C07322=1185.317,71.605,-48.992,-179.176,5.973,148.824
C07323=1185.312,71.854,-49.010,-179.174,5.974,148.823
C07324=1185.308,72.103,-49.027,-179.172,5.975,148.823
C07325=1185.303,72.353,-49.044,-179.168,5.976,148.822
C07326=1185.298,72.602,-49.061,-179.166,5.977,148.822
C07327=1185.293,72.852,-49.078,-179.163,5.978,148.821
C07328=1185.288,73.101,-49.095,-179.161,5.979,148.820
C07329=1185.283,73.350,-49.112,-179.158,5.980,148.820
C07330=1185.279,73.600,-49.129,-179.155,5.981,148.819
C07331=1185.273,73.849,-49.146,-179.153,5.982,148.819
C07332=1185.268,74.098,-49.163,-179.150,5.983,148.818
C07333=1185.263,74.347,-49.181,-179.148,5.984,148.818
C07334=1185.259,74.597,-49.197,-179.145,5.985,148.817
C07335=1185.254,74.847,-49.215,-179.143,5.986,148.817
C07336=1185.249,75.096,-49.231,-179.140,5.987,148.816
C07337=1185.244,75.345,-49.249,-179.137,5.988,148.815
C07338=1185.239,75.594,-49.266,-179.134,5.989,148.815
C07339=1185.234,75.844,-49.283,-179.132,5.990,148.814
C07340=1185.229,76.093,-49.301,-179.129,5.991,148.814
C07341=1185.225,76.343,-49.318,-179.127,5.992,148.813
C07342=1185.219,76.592,-49.335,-179.124,5.993,148.813
C07343=1185.215,76.842,-49.353,-179.122,5.994,148.812
C07344=1185.209,77.090,-49.369,-179.119,5.995,148.812
C07345=1185.205,77.340,-49.387,-179.116,5.996,148.811
C07346=1185.199,77.589,-49.404,-179.113,5.998,148.810
C07347=1185.195,77.839,-49.421,-179.111,5.998,148.810
C07348=1185.190,78.088,-49.439,-179.109,5.999,148.809
C07349=1185.185,78.337,-49.456,-179.105,6.000,148.809
C07350=1185.181,78.587,-49.474,-179.103,6.001,148.808
C07351=1185.175,78.836,-49.491,-179.101,6.002,148.808
C07352=1185.169,79.086,-49.508,-179.098,6.003,148.807
C07353=1185.165,79.334,-49.525,-179.095,6.004,148.807
C07354=1185.160,79.584,-49.542,-179.093,6.006,148.806
C07355=1185.155,79.833,-49.560,-179.090,6.006,148.805
C07356=1185.151,80.083,-49.577,-179.088,6.007,148.805
C07357=1185.146,80.351,-49.596,-179.085,6.009,148.804
C07358=1185.140,80.620,-49.615,-179.081,6.010,148.804
C07359=1185.134,80.888,-49.633,-179.079,6.011,148.803
C07360=1185.129,81.156,-49.653,-179.076,6.012,148.803
C07361=1185.125,81.406,-49.670,-179.073,6.013,148.802
C07362=1185.120,81.655,-49.688,-179.071,6.014,148.802
C07363=1185.115,81.905,-49.705,-179.068,6.015,148.801
C07364=1185.110,82.154,-49.723,-179.066,6.016,148.801
C07365=1185.105,82.403,-49.740,-179.063,6.017,148.800
C07366=1185.100,82.653,-49.757,-179.061,6.018,148.799
C07367=1185.095,82.902,-49.775,-179.057,6.019,148.799
C07368=1185.090,83.152,-49.793,-179.055,6.020,148.798
C07369=1185.086,83.401,-49.810,-179.053,6.021,148.798
C07370=1185.081,83.650,-49.828,-179.050,6.023,148.797
C07371=1185.076,83.900,-49.845,-179.047,6.023,148.797
C07372=1185.071,84.149,-49.863,-179.045,6.025,148.796
C07373=1185.066,84.398,-49.881,-179.042,6.025,148.796
C07374=1185.062,84.647,-49.898,-179.039,6.027,148.795
C07375=1185.057,84.897,-49.916,-179.037,6.028,148.795
C07376=1185.052,85.146,-49.934,-179.034,6.029,148.794
C07377=1185.046,85.396,-49.951,-179.032,6.030,148.794
C07378=1185.042,85.645,-49.969,-179.029,6.031,148.793
C07379=1185.037,85.894,-49.987,-179.026,6.033,148.793
C07380=1185.031,86.144,-50.004,-179.024,6.033,148.792
C07381=1185.027,86.393,-50.022,-179.021,6.035,148.792
C07382=1185.022,86.642,-50.040,-179.018,6.035,148.791
C07383=1185.017,86.891,-50.058,-179.016,6.036,148.790
C07384=1185.012,87.141,-50.075,-179.013,6.038,148.790
C07385=1185.007,87.390,-50.093,-179.011,6.039,148.789
C07386=1185.002,87.639,-50.111,-179.008,6.040,148.789
C07387=1184.997,87.888,-50.129,-179.006,6.041,148.788
C07388=1184.992,88.138,-50.146,-179.002,6.042,148.788
C07389=1184.987,88.387,-50.164,-179.000,6.043,148.787
C07390=1184.982,88.636,-50.182,-178.997,6.044,148.787
C07391=1184.978,88.885,-50.200,-178.995,6.045,148.786
C07392=1184.973,89.134,-50.218,-178.992,6.047,148.786
C07393=1184.968,89.384,-50.235,-178.990,6.048,148.785
C07394=1184.963,89.633,-50.253,-178.987,6.048,148.784
C07395=1184.958,89.883,-50.271,-178.984,6.050,148.784
C07396=1184.954,90.132,-50.289,-178.982,6.050,148.783
C07397=1184.949,90.382,-50.307,-178.979,6.052,148.783
C07398=1184.944,90.631,-50.325,-178.977,6.053,148.783
C07399=1184.939,90.880,-50.343,-178.974,6.054,148.782
C07400=1184.934,91.129,-50.361,-178.971,6.055,148.781
C07401=1184.929,91.378,-50.379,-178.968,6.057,148.781
C07402=1184.924,91.628,-50.396,-178.966,6.058,148.780
C07403=1184.919,91.877,-50.414,-178.963,6.059,148.780
C07404=1184.914,92.126,-50.432,-178.961,6.060,148.779
C07405=1184.910,92.376,-50.451,-178.958,6.061,148.779
C07406=1184.905,92.625,-50.469,-178.955,6.062,148.778
C07407=1184.900,92.875,-50.487,-178.953,6.063,148.778
C07408=1184.895,93.124,-50.505,-178.950,6.065,148.777
C07409=1184.890,93.373,-50.522,-178.948,6.065,148.777
C07410=1184.886,93.622,-50.540,-178.945,6.067,148.776
C07411=1184.880,93.872,-50.559,-178.943,6.068,148.776
C07412=1184.876,94.122,-50.577,-178.939,6.069,148.775
C07413=1184.871,94.371,-50.595,-178.937,6.070,148.775
C07414=1184.866,94.620,-50.613,-178.934,6.071,148.774
C07415=1184.861,94.869,-50.631,-178.932,6.072,148.774
C07416=1184.856,95.118,-50.649,-178.929,6.074,148.773
C07417=1184.851,95.367,-50.667,-178.927,6.075,148.773
C07418=1184.847,95.617,-50.686,-178.924,6.076,148.772
C07419=1184.842,95.866,-50.704,-178.921,6.077,148.771
C07420=1184.836,96.115,-50.723,-178.919,6.079,148.771
C07421=1184.832,96.365,-50.741,-178.916,6.079,148.770
C07422=1184.827,96.614,-50.759,-178.913,6.081,148.770
C07423=1184.822,96.864,-50.777,-178.911,6.081,148.769
C07424=1184.817,97.113,-50.795,-178.908,6.083,148.769
C07425=1184.812,97.362,-50.813,-178.905,6.084,148.768
C07426=1184.808,97.610,-50.832,-178.903,6.085,148.768
C07427=1184.802,97.860,-50.850,-178.900,6.086,148.767
C07428=1184.798,98.110,-50.869,-178.897,6.088,148.767
C07429=1184.793,98.359,-50.887,-178.895,6.089,148.766
C07430=1184.788,98.608,-50.905,-178.892,6.090,148.766
C07431=1184.783,98.857,-50.923,-178.890,6.091,148.765
C07432=1184.778,99.107,-50.942,-178.887,6.092,148.765
C07433=1184.774,99.356,-50.960,-178.884,6.093,148.764
C07434=1184.769,99.605,-50.978,-178.882,6.095,148.764
C07435=1184.764,99.854,-50.996,-178.879,6.095,148.763
C07436=1184.759,100.104,-51.016,-178.876,6.097,148.763
C07437=1184.754,100.353,-51.034,-178.873,6.099,148.762
C07438=1184.749,100.602,-51.052,-178.871,6.099,148.762
C07439=1184.744,100.852,-51.070,-178.868,6.101,148.761
C07440=1184.739,101.101,-51.090,-178.866,6.102,148.761
C07441=1184.735,101.350,-51.108,-178.863,6.104,148.760
C07442=1184.730,101.599,-51.126,-178.860,6.104,148.760
C07443=1184.726,101.849,-51.145,-178.858,6.106,148.759
C07444=1184.720,102.098,-51.163,-178.856,6.107,148.759
C07445=1184.715,102.347,-51.181,-178.852,6.108,148.758
C07446=1184.711,102.597,-51.200,-178.850,6.109,148.758
C07447=1184.705,102.846,-51.219,-178.847,6.110,148.757
C07448=1184.701,103.095,-51.237,-178.845,6.111,148.757
C07449=1184.696,103.344,-51.255,-178.842,6.113,148.756
C07450=1184.691,103.594,-51.274,-178.839,6.114,148.756
C07451=1184.686,103.843,-51.293,-178.837,6.115,148.755
C07452=1184.681,104.092,-51.311,-178.834,6.117,148.755
C07453=1184.676,104.342,-51.330,-178.832,6.118,148.754
C07454=1184.672,104.591,-51.349,-178.829,6.119,148.754
C07455=1184.667,104.840,-51.367,-178.826,6.120,148.753
C07456=1184.662,105.089,-51.386,-178.824,6.122,148.753
C07457=1184.657,105.338,-51.404,-178.821,6.122,148.752
C07458=1184.653,105.588,-51.423,-178.818,6.124,148.752
C07459=1184.647,105.837,-51.442,-178.816,6.125,148.751
C07460=1184.643,106.086,-51.461,-178.813,6.126,148.751
C07461=1184.638,106.355,-51.481,-178.810,6.128,148.750
C07462=1184.633,106.623,-51.501,-178.807,6.129,148.750
C07463=1184.627,106.891,-51.521,-178.804,6.130,148.749
C07464=1184.622,107.160,-51.542,-178.802,6.132,148.749
C07465=1184.617,107.409,-51.560,-178.799,6.133,148.748
C07466=1184.612,107.659,-51.579,-178.796,6.134,148.748
C07467=1184.608,107.908,-51.598,-178.794,6.136,148.747
C07468=1184.603,108.156,-51.617,-178.791,6.136,148.746
C07469=1184.598,108.407,-51.636,-178.788,6.138,148.746
C07470=1184.593,108.655,-51.654,-178.786,6.140,148.746
C07471=1184.588,108.905,-51.673,-178.783,6.140,148.745
C07472=1184.584,109.154,-51.692,-178.780,6.142,148.745
C07473=1184.578,109.403,-51.711,-178.778,6.143,148.744
C07474=1184.574,109.653,-51.729,-178.775,6.144,148.744
C07475=1184.569,109.901,-51.749,-178.773,6.145,148.743
C07476=1184.565,110.151,-51.768,-178.770,6.147,148.743
C07477=1184.559,110.400,-51.786,-178.767,6.148,148.742
C07478=1184.554,110.649,-51.805,-178.765,6.149,148.742
C07479=1184.550,110.898,-51.825,-178.762,6.151,148.741
C07480=1184.545,111.147,-51.843,-178.759,6.152,148.741
C07481=1184.540,111.397,-51.862,-178.757,6.153,148.740
C07482=1184.535,111.646,-51.882,-178.754,6.155,148.740
C07483=1184.530,111.896,-51.900,-178.751,6.156,148.739
C07484=1184.525,112.145,-51.919,-178.749,6.157,148.739
C07485=1184.521,112.394,-51.938,-178.746,6.158,148.738
C07486=1184.516,112.643,-51.958,-178.743,6.160,148.738
C07487=1184.511,112.893,-51.976,-178.741,6.161,148.737
C07488=1184.506,113.142,-51.995,-178.738,6.162,148.737
C07489=1184.501,113.391,-52.015,-178.735,6.164,148.736
C07490=1184.497,113.640,-52.034,-178.733,6.164,148.736
C07491=1184.492,113.889,-52.053,-178.730,6.166,148.735
C07492=1184.487,114.138,-52.071,-178.727,6.168,148.735
C07493=1184.482,114.388,-52.091,-178.725,6.168,148.734
C07494=1184.477,114.637,-52.110,-178.722,6.170,148.734
C07495=1184.473,114.886,-52.129,-178.719,6.172,148.733
C07496=1184.468,115.135,-52.149,-178.717,6.172,148.733
C07497=1184.463,115.385,-52.168,-178.714,6.174,148.732
C07498=1184.458,115.634,-52.186,-178.712,6.175,148.732
C07499=1184.453,115.883,-52.206,-178.709,6.176,148.731
C07500=1184.448,116.132,-52.225,-178.706,6.178,148.731
C07501=1184.444,116.381,-52.244,-178.704,6.179,148.731
C07502=1184.438,116.630,-52.264,-178.701,6.181,148.730
C07503=1184.434,116.880,-52.283,-178.698,6.182,148.730
C07504=1184.428,117.129,-52.302,-178.696,6.183,148.729
C07505=1184.424,117.378,-52.322,-178.693,6.185,148.729
C07506=1184.420,117.628,-52.341,-178.691,6.185,148.728
C07507=1184.414,117.876,-52.360,-178.688,6.187,148.728
C07508=1184.410,118.126,-52.380,-178.685,6.189,148.727
C07509=1184.405,118.375,-52.399,-178.683,6.190,148.727
C07510=1184.400,118.624,-52.418,-178.680,6.191,148.726
C07511=1184.395,118.874,-52.438,-178.677,6.193,148.726
C07512=1184.391,119.122,-52.457,-178.675,6.194,148.725
C07513=1184.386,119.372,-52.476,-178.672,6.195,148.725
C07514=1184.381,119.621,-52.496,-178.669,6.197,148.724
C07515=1184.376,119.870,-52.515,-178.667,6.198,148.724
C07516=1184.371,120.120,-52.535,-178.664,6.199,148.723
C07517=1184.367,120.368,-52.554,-178.661,6.201,148.723
C07518=1184.362,120.618,-52.573,-178.658,6.202,148.722
C07519=1184.357,120.867,-52.593,-178.656,6.203,148.722
C07520=1184.352,121.116,-52.612,-178.653,6.205,148.722
C07521=1184.347,121.366,-52.632,-178.650,6.206,148.721
C07522=1184.343,121.614,-52.651,-178.648,6.208,148.721
C07523=1184.338,121.863,-52.671,-178.645,6.209,148.720
C07524=1184.333,122.113,-52.691,-178.643,6.210,148.720
C07525=1184.328,122.362,-52.710,-178.640,6.212,148.719
C07526=1184.323,122.611,-52.730,-178.637,6.213,148.719
C07527=1184.318,122.861,-52.749,-178.635,6.214,148.718
C07528=1184.313,123.110,-52.769,-178.632,6.216,148.718
C07529=1184.309,123.358,-52.788,-178.629,6.217,148.717
C07530=1184.305,123.608,-52.808,-178.627,6.218,148.717
C07531=1184.299,123.857,-52.827,-178.624,6.220,148.716
C07532=1184.295,124.106,-52.847,-178.621,6.221,148.716
C07533=1184.290,124.355,-52.867,-178.619,6.222,148.715
C07534=1184.285,124.604,-52.887,-178.616,6.224,148.715
C07535=1184.280,124.854,-52.906,-178.613,6.226,148.714
C07536=1184.275,125.103,-52.926,-178.611,6.226,148.714
C07537=1184.271,125.352,-52.946,-178.608,6.228,148.714
C07538=1184.266,125.601,-52.966,-178.606,6.230,148.713
C07539=1184.261,125.851,-52.985,-178.603,6.231,148.713
C07540=1184.256,126.100,-53.005,-178.600,6.232,148.712
C07541=1184.252,126.348,-53.024,-178.598,6.234,148.712
C07542=1184.247,126.598,-53.044,-178.595,6.235,148.711
C07543=1184.242,126.847,-53.064,-178.592,6.236,148.711
C07544=1184.238,127.096,-53.084,-178.590,6.238,148.710
C07545=1184.232,127.345,-53.103,-178.587,6.240,148.710
C07546=1184.228,127.595,-53.123,-178.584,6.240,148.709
C07547=1184.223,127.844,-53.143,-178.582,6.242,148.709
C07548=1184.219,128.093,-53.163,-178.579,6.244,148.709
C07549=1184.214,128.342,-53.183,-178.577,6.245,148.708
C07550=1184.209,128.591,-53.203,-178.574,6.246,148.708
C07551=1184.204,128.841,-53.222,-178.571,6.248,148.707
C07552=1184.200,129.090,-53.243,-178.568,6.250,148.707
C07553=1184.194,129.340,-53.263,-178.566,6.251,148.706
C07554=1184.189,129.588,-53.283,-178.563,6.252,148.706
C07555=1184.184,129.837,-53.303,-178.560,6.254,148.705
C07556=1184.180,130.086,-53.323,-178.558,6.255,148.705
C07557=1184.175,130.336,-53.343,-178.555,6.257,148.705
C07558=1184.171,130.585,-53.363,-178.552,6.258,148.704
C07559=1184.165,130.834,-53.382,-178.549,6.260,148.704
C07560=1184.161,131.083,-53.403,-178.547,6.261,148.703
C07561=1184.156,131.332,-53.422,-178.545,6.262,148.703
C07562=1184.152,131.581,-53.443,-178.541,6.264,148.702
C07563=1184.147,131.831,-53.462,-178.539,6.265,148.702
C07564=1184.141,132.079,-53.483,-178.537,6.266,148.701
C07565=1184.136,132.348,-53.504,-178.533,6.268,148.701
C07566=1184.131,132.618,-53.526,-178.531,6.270,148.700
C07567=1184.127,132.886,-53.548,-178.528,6.271,148.700
C07568=1184.121,133.155,-53.570,-178.525,6.273,148.699
C07569=1184.116,133.403,-53.590,-178.522,6.275,148.699
C07570=1184.111,133.652,-53.609,-178.519,6.276,148.699
C07571=1184.107,133.901,-53.630,-178.517,6.277,148.698
C07572=1184.102,134.150,-53.650,-178.514,6.279,148.698
C07573=1184.098,134.400,-53.670,-178.511,6.280,148.697
C07574=1184.092,134.649,-53.691,-178.509,6.281,148.697
C07575=1184.088,134.898,-53.711,-178.507,6.283,148.696
C07576=1184.083,135.148,-53.731,-178.503,6.284,148.696
C07577=1184.078,135.396,-53.751,-178.501,6.286,148.695
C07578=1184.073,135.645,-53.772,-178.498,6.288,148.695
C07579=1184.068,135.895,-53.791,-178.496,6.289,148.695
C07580=1184.064,136.144,-53.812,-178.493,6.291,148.694
C07581=1184.059,136.393,-53.832,-178.490,6.292,148.694
C07582=1184.054,136.642,-53.853,-178.487,6.294,148.693
C07583=1184.050,136.891,-53.873,-178.485,6.295,148.693
C07584=1184.045,137.140,-53.893,-178.483,6.297,148.692
C07585=1184.041,137.389,-53.913,-178.479,6.298,148.692
C07586=1184.035,137.639,-53.934,-178.477,6.300,148.691
C07587=1184.031,137.888,-53.955,-178.475,6.301,148.691
C07588=1184.026,138.137,-53.974,-178.472,6.302,148.691
C07589=1184.022,138.386,-53.995,-178.469,6.304,148.690
C07590=1184.016,138.635,-54.015,-178.466,6.306,148.690
C07591=1184.012,138.884,-54.036,-178.464,6.306,148.689
C07592=1184.007,139.133,-54.056,-178.461,6.308,148.689
C07593=1184.002,139.382,-54.077,-178.459,6.310,148.688
C07594=1183.997,139.631,-54.097,-178.456,6.312,148.688
C07595=1183.993,139.880,-54.117,-178.453,6.313,148.687
C07596=1183.988,140.130,-54.138,-178.451,6.314,148.687
C07597=1183.983,140.379,-54.158,-178.448,6.316,148.687
C07598=1183.978,140.628,-54.179,-178.445,6.318,148.686
C07599=1183.974,140.877,-54.200,-178.442,6.319,148.686
C07600=1183.969,141.126,-54.220,-178.440,6.321,148.686
C07601=1183.964,141.375,-54.241,-178.437,6.322,148.685
C07602=1183.960,141.624,-54.262,-178.434,6.323,148.684
C07603=1183.955,141.873,-54.282,-178.432,6.325,148.684
C07604=1183.950,142.122,-54.303,-178.429,6.327,148.684
C07605=1183.946,142.371,-54.323,-178.426,6.329,148.683
C07606=1183.940,142.620,-54.344,-178.424,6.329,148.683
C07607=1183.936,142.869,-54.365,-178.421,6.331,148.682
C07608=1183.931,143.119,-54.386,-178.418,6.333,148.682
C07609=1183.926,143.367,-54.406,-178.416,6.335,148.682
C07610=1183.922,143.616,-54.426,-178.413,6.336,148.681
C07611=1183.917,143.866,-54.448,-178.411,6.337,148.681
C07612=1183.913,144.115,-54.468,-178.408,6.339,148.680
C07613=1183.908,144.365,-54.489,-178.405,6.341,148.680
C07614=1183.903,144.614,-54.509,-178.402,6.342,148.679
C07615=1183.898,144.863,-54.530,-178.400,6.344,148.679
C07616=1183.894,145.112,-54.551,-178.397,6.346,148.679
C07617=1183.888,145.361,-54.572,-178.395,6.347,148.678
C07618=1183.884,145.610,-54.592,-178.392,6.348,148.678
C07619=1183.879,145.859,-54.613,-178.389,6.350,148.677
C07620=1183.875,146.108,-54.634,-178.386,6.352,148.677
C07621=1183.870,146.357,-54.655,-178.384,6.353,148.676
C07622=1183.865,146.606,-54.675,-178.382,6.354,148.676
C07623=1183.860,146.855,-54.696,-178.379,6.356,148.676
C07624=1183.855,147.105,-54.718,-178.376,6.358,148.675
C07625=1183.851,147.354,-54.738,-178.373,6.359,148.675
C07626=1183.846,147.603,-54.760,-178.370,6.361,148.674
C07627=1183.842,147.852,-54.780,-178.368,6.363,148.674
C07628=1183.836,148.101,-54.801,-178.365,6.364,148.674
C07629=1183.832,148.350,-54.821,-178.363,6.366,148.673
C07630=1183.827,148.598,-54.843,-178.360,6.367,148.673
C07631=1183.822,148.848,-54.864,-178.357,6.369,148.672
C07632=1183.818,149.097,-54.885,-178.355,6.371,148.672
C07633=1183.813,149.347,-54.906,-178.352,6.372,148.671
C07634=1183.809,149.595,-54.927,-178.349,6.374,148.671
C07635=1183.804,149.844,-54.948,-178.347,6.375,148.671
C07636=1183.798,150.093,-54.969,-178.344,6.377,148.670
C07637=1183.794,150.342,-54.990,-178.341,6.378,148.670
C07638=1183.790,150.592,-55.011,-178.339,6.380,148.670
C07639=1183.785,150.841,-55.032,-178.336,6.382,148.669
C07640=1183.780,151.089,-55.053,-178.333,6.384,148.669
C07641=1183.775,151.339,-55.074,-178.330,6.385,148.668
C07642=1183.770,151.588,-55.095,-178.328,6.386,148.668
C07643=1183.765,151.836,-55.117,-178.325,6.388,148.667
C07644=1183.761,152.086,-55.138,-178.323,6.390,148.667
C07645=1183.757,152.335,-55.159,-178.320,6.391,148.667
C07646=1183.751,152.584,-55.180,-178.317,6.393,148.666
C07647=1183.747,152.833,-55.201,-178.315,6.395,148.666
C07648=1183.742,153.082,-55.222,-178.312,6.397,148.666
C07649=1183.737,153.332,-55.244,-178.309,6.399,148.665
C07650=1183.733,153.580,-55.265,-178.307,6.399,148.665
C07651=1183.728,153.829,-55.286,-178.304,6.401,148.664
C07652=1183.723,154.078,-55.307,-178.301,6.403,148.664
C07653=1183.719,154.328,-55.329,-178.299,6.404,148.663
C07654=1183.714,154.576,-55.350,-178.296,6.406,148.663
C07655=1183.709,154.825,-55.371,-178.293,6.408,148.663
C07656=1183.705,155.074,-55.393,-178.291,6.410,148.662
C07657=1183.700,155.324,-55.414,-178.288,6.411,148.662
C07658=1183.695,155.573,-55.436,-178.285,6.413,148.662
C07659=1183.690,155.822,-55.456,-178.283,6.414,148.661
C07660=1183.686,156.070,-55.478,-178.280,6.416,148.661
C07661=1183.682,156.319,-55.500,-178.277,6.417,148.660
C07662=1183.676,156.569,-55.521,-178.275,6.419,148.660
C07663=1183.671,156.817,-55.542,-178.272,6.421,148.659
C07664=1183.667,157.067,-55.564,-178.269,6.423,148.659
C07665=1183.662,157.316,-55.585,-178.266,6.424,148.659
C07666=1183.657,157.565,-55.607,-178.264,6.426,148.658
C07667=1183.653,157.814,-55.627,-178.261,6.428,148.658
C07668=1183.648,158.063,-55.649,-178.258,6.430,148.658
C07669=1183.643,158.332,-55.673,-178.256,6.432,148.657
C07670=1183.638,158.601,-55.696,-178.253,6.433,148.657
C07671=1183.633,158.870,-55.720,-178.250,6.435,148.656
C07672=1183.628,159.138,-55.742,-178.247,6.436,148.656
C07673=1183.623,159.388,-55.764,-178.245,6.438,148.655
C07674=1183.618,159.637,-55.785,-178.242,6.440,148.655
C07675=1183.613,159.886,-55.807,-178.239,6.442,148.655
C07676=1183.609,160.135,-55.829,-178.236,6.444,148.654
C07677=1183.604,160.384,-55.850,-178.234,6.445,148.654
C07678=1183.600,160.634,-55.872,-178.231,6.447,148.654
C07679=1183.595,160.882,-55.893,-178.228,6.449,148.653
C07680=1183.590,161.131,-55.915,-178.225,6.450,148.653
C07681=1183.586,161.380,-55.937,-178.223,6.451,148.652
C07682=1183.581,161.629,-55.959,-178.220,6.453,148.652
C07683=1183.576,161.878,-55.980,-178.218,6.455,148.651
C07684=1183.571,162.127,-56.002,-178.215,6.457,148.651
C07685=1183.566,162.376,-56.024,-178.212,6.458,148.651
C07686=1183.562,162.625,-56.046,-178.210,6.460,148.650
C07687=1183.557,162.874,-56.067,-178.207,6.462,148.650
C07688=1183.552,163.123,-56.089,-178.204,6.464,148.650
C07689=1183.548,163.372,-56.111,-178.202,6.465,148.649
C07690=1183.543,163.621,-56.132,-178.199,6.467,148.649
C07691=1183.539,163.871,-56.154,-178.196,6.469,148.649
C07692=1183.534,164.119,-56.176,-178.194,6.471,148.648
C07693=1183.529,164.368,-56.197,-178.191,6.473,148.648
C07694=1183.525,164.617,-56.219,-178.188,6.474,148.647
C07695=1183.520,164.866,-56.241,-178.186,6.476,148.647
C07696=1183.516,165.115,-56.263,-178.183,6.478,148.647
C07697=1183.511,165.364,-56.285,-178.180,6.480,148.646
C07698=1183.506,165.613,-56.307,-178.178,6.481,148.646
C07699=1183.502,165.862,-56.329,-178.175,6.483,148.646
C07700=1183.497,166.112,-56.351,-178.173,6.484,148.645
C07701=1183.492,166.360,-56.373,-178.170,6.486,148.645
C07702=1183.487,166.610,-56.395,-178.167,6.488,148.644
C07703=1183.483,166.858,-56.417,-178.165,6.489,148.644
C07704=1183.478,167.108,-56.439,-178.162,6.491,148.644
C07705=1183.473,167.356,-56.460,-178.159,6.493,148.643
C07706=1183.469,167.605,-56.482,-178.157,6.495,148.643
C07707=1183.464,167.854,-56.505,-178.154,6.497,148.643
C07708=1183.459,168.102,-56.527,-178.151,6.498,148.642
C07709=1183.455,168.352,-56.549,-178.149,6.500,148.642
C07710=1183.450,168.600,-56.571,-178.146,6.502,148.641
C07711=1183.446,168.850,-56.593,-178.143,6.504,148.641
C07712=1183.441,169.099,-56.616,-178.141,6.505,148.641
C07713=1183.436,169.348,-56.637,-178.138,6.507,148.640
C07714=1183.431,169.597,-56.659,-178.135,6.509,148.640
C07715=1183.427,169.846,-56.681,-178.133,6.511,148.640
C07716=1183.423,170.095,-56.704,-178.130,6.513,148.639
C07717=1183.417,170.344,-56.726,-178.127,6.514,148.639
C07718=1183.413,170.593,-56.748,-178.125,6.516,148.639
C07719=1183.408,170.842,-56.770,-178.122,6.518,148.638
C07720=1183.404,171.091,-56.792,-178.119,6.520,148.638
C07721=1183.398,171.339,-56.815,-178.117,6.521,148.637
C07722=1183.394,171.589,-56.837,-178.114,6.523,148.637
C07723=1183.389,171.837,-56.858,-178.111,6.525,148.637
C07724=1183.385,172.086,-56.882,-178.108,6.527,148.636
C07725=1183.380,172.336,-56.904,-178.106,6.529,148.636
C07726=1183.375,172.584,-56.926,-178.103,6.530,148.636
C07727=1183.370,172.834,-56.948,-178.100,6.532,148.635
C07728=1183.366,173.082,-56.971,-178.098,6.534,148.635
C07729=1183.362,173.331,-56.993,-178.095,6.536,148.635
C07730=1183.357,173.581,-57.015,-178.092,6.537,148.634
C07731=1183.352,173.829,-57.038,-178.090,6.539,148.634
C07732=1183.348,174.078,-57.060,-178.087,6.541,148.633
C07733=1183.342,174.327,-57.082,-178.084,6.543,148.633
C07734=1183.338,174.576,-57.105,-178.082,6.545,148.633
C07735=1183.334,174.825,-57.127,-178.079,6.546,148.632
C07736=1183.329,175.074,-57.150,-178.076,6.548,148.632
C07737=1183.324,175.323,-57.172,-178.074,6.550,148.632
C07738=1183.319,175.573,-57.195,-178.071,6.552,148.631
C07739=1183.315,175.821,-57.217,-178.068,6.553,148.631
C07740=1183.310,176.070,-57.239,-178.066,6.555,148.631
C07741=1183.305,176.318,-57.262,-178.063,6.557,148.630
C07742=1183.301,176.568,-57.284,-178.060,6.560,148.630
C07743=1183.296,176.817,-57.307,-178.058,6.562,148.630
C07744=1183.291,177.065,-57.329,-178.055,6.564,148.629
C07745=1183.287,177.314,-57.352,-178.052,6.565,148.629
C07746=1183.282,177.564,-57.374,-178.050,6.567,148.629
C07747=1183.278,177.812,-57.397,-178.047,6.569,148.628
C07748=1183.273,178.061,-57.419,-178.044,6.571,148.628
C07749=1183.269,178.310,-57.442,-178.042,6.572,148.628
C07750=1183.264,178.560,-57.465,-178.039,6.574,148.627
C07751=1183.259,178.808,-57.487,-178.036,6.576,148.627
C07752=1183.255,179.057,-57.511,-178.033,6.578,148.626
C07753=1183.250,179.306,-57.533,-178.031,6.580,148.626
C07754=1183.245,179.555,-57.556,-178.028,6.581,148.626
C07755=1183.241,179.804,-57.578,-178.025,6.583,148.625
C07756=1183.236,180.053,-57.601,-178.023,6.585,148.625
C07757=1183.232,180.302,-57.624,-178.021,6.587,148.625
C07758=1183.226,180.551,-57.646,-178.018,6.589,148.625
C07759=1183.222,180.800,-57.669,-178.015,6.591,148.624
C07760=1183.218,181.048,-57.692,-178.013,6.592,148.624
C07761=1183.213,181.298,-57.715,-178.009,6.595,148.623
C07762=1183.208,181.546,-57.737,-178.007,6.597,148.623
C07763=1183.204,181.795,-57.761,-178.004,6.599,148.623
C07764=1183.199,182.044,-57.783,-178.001,6.600,148.622
C07765=1183.195,182.293,-57.806,-177.999,6.602,148.622
C07766=1183.189,182.542,-57.829,-177.996,6.604,148.622
C07767=1183.185,182.791,-57.852,-177.994,6.606,148.622
C07768=1183.180,183.040,-57.874,-177.991,6.608,148.621
C07769=1183.176,183.289,-57.897,-177.988,6.610,148.621
C07770=1183.172,183.538,-57.921,-177.986,6.611,148.620
C07771=1183.166,183.786,-57.944,-177.983,6.613,148.620
C07772=1183.162,184.035,-57.966,-177.980,6.615,148.620
C07773=1183.157,184.305,-57.991,-177.977,6.618,148.619
C07774=1183.152,184.575,-58.016,-177.975,6.619,148.619
C07775=1183.147,184.844,-58.041,-177.972,6.621,148.619
C07776=1183.142,185.114,-58.066,-177.969,6.624,148.618
C07777=1183.137,185.363,-58.089,-177.966,6.626,148.618
C07778=1183.133,185.611,-58.112,-177.963,6.627,148.618
C07779=1183.128,185.861,-58.135,-177.961,6.629,148.617
C07780=1183.123,186.109,-58.158,-177.958,6.631,148.617
C07781=1183.119,186.358,-58.180,-177.956,6.633,148.617
C07782=1183.114,186.607,-58.204,-177.953,6.635,148.616
C07783=1183.109,186.856,-58.227,-177.950,6.637,148.616
C07784=1183.105,187.105,-58.250,-177.947,6.639,148.616
C07785=1183.101,187.354,-58.273,-177.944,6.641,148.615
C07786=1183.096,187.603,-58.297,-177.942,6.643,148.615
C07787=1183.091,187.852,-58.320,-177.939,6.645,148.615
C07788=1183.086,188.100,-58.343,-177.936,6.646,148.614
C07789=1183.082,188.349,-58.366,-177.934,6.648,148.614
C07790=1183.077,188.598,-58.389,-177.932,6.650,148.614
C07791=1183.073,188.847,-58.412,-177.929,6.652,148.614
C07792=1183.068,189.096,-58.436,-177.926,6.655,148.613
C07793=1183.063,189.345,-58.459,-177.923,6.656,148.613
C07794=1183.059,189.594,-58.482,-177.920,6.658,148.613
C07795=1183.055,189.843,-58.505,-177.918,6.660,148.612
C07796=1183.050,190.091,-58.529,-177.915,6.662,148.612
C07797=1183.045,190.340,-58.552,-177.913,6.664,148.612
C07798=1183.040,190.589,-58.576,-177.910,6.666,148.611
C07799=1183.036,190.838,-58.599,-177.907,6.668,148.611
C07800=1183.031,191.087,-58.622,-177.904,6.670,148.611
C07801=1183.027,191.336,-58.645,-177.902,6.672,148.610
C07802=1183.022,191.585,-58.669,-177.899,6.674,148.610
C07803=1183.018,191.834,-58.692,-177.897,6.676,148.610
C07804=1183.013,192.082,-58.716,-177.894,6.678,148.609
C07805=1183.008,192.331,-58.739,-177.891,6.679,148.609
C07806=1183.004,192.580,-58.763,-177.888,6.682,148.609
C07807=1182.999,192.829,-58.786,-177.885,6.684,148.608
C07808=1182.994,193.078,-58.809,-177.883,6.686,148.608
C07809=1182.990,193.327,-58.833,-177.881,6.688,148.608
C07810=1182.985,193.576,-58.857,-177.878,6.690,148.608
C07811=1182.981,193.825,-58.880,-177.875,6.691,148.607
C07812=1182.976,194.074,-58.904,-177.873,6.693,148.607
C07813=1182.971,194.322,-58.928,-177.870,6.696,148.607
C07814=1182.967,194.571,-58.951,-177.867,6.698,148.606
C07815=1182.962,194.820,-58.974,-177.865,6.700,148.606
C07816=1182.958,195.069,-58.998,-177.862,6.701,148.606
C07817=1182.953,195.318,-59.022,-177.859,6.703,148.605
C07818=1182.948,195.567,-59.045,-177.857,6.705,148.605
C07819=1182.944,195.815,-59.069,-177.854,6.708,148.605
C07820=1182.939,196.064,-59.093,-177.851,6.710,148.605
C07821=1182.934,196.313,-59.116,-177.848,6.712,148.604
C07822=1182.930,196.562,-59.140,-177.846,6.713,148.604
C07823=1182.925,196.811,-59.163,-177.843,6.715,148.604
C07824=1182.921,197.060,-59.187,-177.841,6.717,148.603
C07825=1182.916,197.308,-59.211,-177.838,6.720,148.603
C07826=1182.912,197.557,-59.234,-177.835,6.722,148.603
C07827=1182.907,197.805,-59.258,-177.832,6.723,148.602
C07828=1182.902,198.054,-59.282,-177.830,6.725,148.602
C07829=1182.898,198.303,-59.306,-177.828,6.727,148.602
C07830=1182.893,198.552,-59.329,-177.824,6.730,148.602
C07831=1182.890,198.801,-59.353,-177.822,6.732,148.601
C07832=1182.885,199.050,-59.377,-177.819,6.734,148.601
C07833=1182.880,199.299,-59.402,-177.817,6.736,148.601
C07834=1182.875,199.548,-59.425,-177.814,6.738,148.600
C07835=1182.871,199.796,-59.449,-177.811,6.740,148.600
C07836=1182.866,200.045,-59.472,-177.808,6.742,148.600
C07837=1182.862,200.294,-59.496,-177.806,6.744,148.599
C07838=1182.857,200.543,-59.520,-177.803,6.746,148.599
C07839=1182.852,200.791,-59.544,-177.801,6.748,148.599
C07840=1182.848,201.041,-59.568,-177.797,6.750,148.599
C07841=1182.843,201.290,-59.592,-177.795,6.752,148.598
C07842=1182.839,201.538,-59.616,-177.793,6.754,148.598
C07843=1182.834,201.787,-59.640,-177.790,6.756,148.598
C07844=1182.830,202.035,-59.664,-177.787,6.758,148.597
C07845=1182.825,202.284,-59.688,-177.784,6.760,148.597
C07846=1182.820,202.533,-59.712,-177.782,6.763,148.597
C07847=1182.816,202.782,-59.736,-177.779,6.764,148.597
C07848=1182.812,203.031,-59.760,-177.777,6.766,148.596
C07849=1182.806,203.280,-59.784,-177.773,6.769,148.596
C07850=1182.802,203.528,-59.808,-177.771,6.771,148.596
C07851=1182.798,203.777,-59.832,-177.768,6.773,148.596
C07852=1182.793,204.026,-59.856,-177.766,6.775,148.595
C07853=1182.788,204.275,-59.881,-177.763,6.776,148.595
C07854=1182.784,204.524,-59.905,-177.760,6.779,148.595
C07855=1182.780,204.772,-59.929,-177.758,6.781,148.594
C07856=1182.775,205.021,-59.953,-177.755,6.783,148.594
C07857=1182.770,205.270,-59.977,-177.752,6.785,148.594
C07858=1182.766,205.519,-60.001,-177.750,6.788,148.594
C07859=1182.761,205.767,-60.025,-177.747,6.789,148.593
C07860=1182.756,206.016,-60.050,-177.744,6.791,148.593
C07861=1182.752,206.265,-60.074,-177.742,6.793,148.593
C07862=1182.748,206.514,-60.098,-177.739,6.796,148.593
C07863=1182.743,206.763,-60.123,-177.736,6.798,148.592
C07864=1182.738,207.011,-60.147,-177.734,6.800,148.592
C07865=1182.734,207.260,-60.171,-177.731,6.802,148.592
C07866=1182.729,207.509,-60.196,-177.728,6.804,148.591
C07867=1182.725,207.758,-60.220,-177.725,6.806,148.591
C07868=1182.720,208.006,-60.245,-177.723,6.808,148.591
C07869=1182.716,208.255,-60.269,-177.721,6.810,148.591
C07870=1182.712,208.504,-60.293,-177.717,6.813,148.590
C07871=1182.706,208.753,-60.317,-177.715,6.814,148.590
C07872=1182.702,209.002,-60.341,-177.713,6.817,148.590
C07873=1182.697,209.250,-60.366,-177.710,6.818,148.589
C07874=1182.693,209.500,-60.390,-177.707,6.821,148.589
C07875=1182.688,209.748,-60.415,-177.705,6.823,148.589
C07876=1182.683,209.997,-60.439,-177.702,6.825,148.589
C07877=1182.679,210.268,-60.466,-177.699,6.828,148.588
C07878=1182.674,210.538,-60.493,-177.696,6.829,148.588
C07879=1182.669,210.808,-60.519,-177.693,6.832,148.588
C07880=1182.663,211.078,-60.546,-177.690,6.834,148.587
C07881=1182.660,211.327,-60.571,-177.687,6.837,148.587
C07882=1182.654,211.576,-60.595,-177.685,6.839,148.587
C07883=1182.650,211.824,-60.619,-177.682,6.840,148.587
C07884=1182.646,212.074,-60.644,-177.679,6.843,148.587
C07885=1182.641,212.322,-60.668,-177.677,6.845,148.586
C07886=1182.636,212.571,-60.693,-177.674,6.847,148.586
C07887=1182.632,212.820,-60.718,-177.672,6.849,148.586
C07888=1182.627,213.068,-60.743,-177.669,6.852,148.585
C07889=1182.624,213.317,-60.767,-177.666,6.854,148.585
C07890=1182.618,213.566,-60.792,-177.664,6.856,148.585
C07891=1182.613,213.815,-60.817,-177.660,6.858,148.585
C07892=1182.610,214.064,-60.841,-177.658,6.860,148.584
C07893=1182.605,214.312,-60.867,-177.656,6.862,148.584
C07894=1182.600,214.560,-60.891,-177.653,6.864,148.584
C07895=1182.596,214.810,-60.916,-177.650,6.867,148.584
C07896=1182.591,215.058,-60.940,-177.648,6.869,148.583
C07897=1182.587,215.307,-60.965,-177.645,6.871,148.583
C07898=1182.582,215.556,-60.990,-177.642,6.873,148.583
C07899=1182.578,215.804,-61.014,-177.639,6.875,148.583
C07900=1182.573,216.053,-61.039,-177.637,6.877,148.582
C07901=1182.568,216.302,-61.065,-177.634,6.880,148.582
C07902=1182.565,216.551,-61.089,-177.631,6.882,148.582
C07903=1182.559,216.799,-61.114,-177.629,6.884,148.582
C07904=1182.555,217.048,-61.139,-177.626,6.886,148.581
C07905=1182.551,217.297,-61.164,-177.623,6.889,148.581
C07906=1182.546,217.546,-61.189,-177.621,6.890,148.581
C07907=1182.541,217.794,-61.214,-177.618,6.893,148.581
C07908=1182.537,218.043,-61.238,-177.615,6.895,148.580
C07909=1182.533,218.291,-61.264,-177.613,6.897,148.580
C07910=1182.528,218.540,-61.288,-177.610,6.900,148.580
C07911=1182.523,218.790,-61.313,-177.607,6.902,148.580
C07912=1182.519,219.037,-61.338,-177.605,6.903,148.579
C07913=1182.515,219.287,-61.363,-177.602,6.906,148.579
C07914=1182.510,219.535,-61.389,-177.599,6.908,148.579
C07915=1182.505,219.784,-61.414,-177.597,6.910,148.579
C07916=1182.501,220.032,-61.439,-177.594,6.913,148.579
C07917=1182.497,220.282,-61.464,-177.591,6.915,148.578
C07918=1182.492,220.530,-61.489,-177.589,6.917,148.578
C07919=1182.487,220.779,-61.514,-177.586,6.920,148.578
C07920=1182.482,221.027,-61.539,-177.583,6.921,148.577
C07921=1182.479,221.276,-61.564,-177.581,6.924,148.577
C07922=1182.474,221.524,-61.589,-177.578,6.926,148.577
C07923=1182.469,221.774,-61.614,-177.576,6.928,148.577
C07924=1182.465,222.023,-61.640,-177.573,6.930,148.577
C07925=1182.460,222.271,-61.665,-177.570,6.933,148.576
C07926=1182.456,222.520,-61.690,-177.567,6.935,148.576
C07927=1182.452,222.768,-61.715,-177.565,6.937,148.576
C07928=1182.447,223.017,-61.740,-177.562,6.940,148.576
C07929=1182.442,223.265,-61.766,-177.559,6.941,148.575
C07930=1182.438,223.514,-61.791,-177.557,6.944,148.575
C07931=1182.433,223.763,-61.816,-177.554,6.946,148.575
C07932=1182.429,224.012,-61.842,-177.551,6.948,148.575
C07933=1182.424,224.261,-61.868,-177.549,6.950,148.575
C07934=1182.419,224.509,-61.892,-177.546,6.953,148.574
C07935=1182.415,224.758,-61.918,-177.544,6.955,148.574
C07936=1182.411,225.006,-61.943,-177.541,6.958,148.574
C07937=1182.407,225.255,-61.969,-177.538,6.960,148.574
C07938=1182.402,225.504,-61.994,-177.536,6.962,148.573
C07939=1182.397,225.752,-62.019,-177.532,6.964,148.573
C07940=1182.393,226.001,-62.045,-177.530,6.966,148.573
C07941=1182.388,226.249,-62.070,-177.528,6.968,148.573
C07942=1182.384,226.499,-62.095,-177.525,6.971,148.573
C07943=1182.380,226.747,-62.121,-177.522,6.973,148.572
C07944=1182.375,226.995,-62.146,-177.520,6.976,148.572
C07945=1182.370,227.244,-62.172,-177.517,6.978,148.572
C07946=1182.366,227.493,-62.198,-177.515,6.980,148.572
C07947=1182.361,227.741,-62.223,-177.511,6.982,148.571
C07948=1182.357,227.990,-62.249,-177.509,6.984,148.571
C07949=1182.352,228.239,-62.274,-177.507,6.986,148.571
C07950=1182.348,228.488,-62.299,-177.503,6.989,148.571
C07951=1182.344,228.736,-62.325,-177.501,6.991,148.571
C07952=1182.339,228.984,-62.350,-177.498,6.994,148.570
C07953=1182.335,229.233,-62.376,-177.496,6.996,148.570
C07954=1182.330,229.482,-62.403,-177.493,6.998,148.570
C07955=1182.325,229.731,-62.428,-177.490,7.001,148.570
C07956=1182.321,229.979,-62.454,-177.488,7.003,148.570
C07957=1182.316,230.228,-62.479,-177.485,7.006,148.569
C07958=1182.312,230.477,-62.505,-177.482,7.007,148.569
C07959=1182.307,230.725,-62.531,-177.480,7.010,148.569
C07960=1182.303,230.974,-62.556,-177.477,7.012,148.569
C07961=1182.299,231.223,-62.582,-177.475,7.014,148.569
C07962=1182.294,231.471,-62.607,-177.472,7.017,148.568
C07963=1182.289,231.720,-62.634,-177.469,7.019,148.568
C07964=1182.285,231.969,-62.660,-177.466,7.022,148.568
C07965=1182.281,232.217,-62.685,-177.464,7.024,148.568
C07966=1182.276,232.466,-62.711,-177.461,7.026,148.567
C07967=1182.272,232.714,-62.736,-177.459,7.029,148.567
C07968=1182.267,232.963,-62.762,-177.456,7.030,148.567
C07969=1182.262,233.212,-62.789,-177.453,7.033,148.567
C07970=1182.258,233.460,-62.815,-177.451,7.035,148.567
C07971=1182.254,233.709,-62.840,-177.448,7.037,148.567
C07972=1182.249,233.957,-62.866,-177.445,7.040,148.566
C07973=1182.245,234.206,-62.892,-177.443,7.042,148.566
C07974=1182.240,234.455,-62.918,-177.440,7.045,148.566
C07975=1182.235,234.703,-62.944,-177.438,7.047,148.566
C07976=1182.231,234.952,-62.970,-177.434,7.050,148.566
C07977=1182.227,235.200,-62.996,-177.432,7.052,148.565
C07978=1182.222,235.449,-63.022,-177.429,7.054,148.565
C07979=1182.218,235.698,-63.048,-177.427,7.057,148.565
C07980=1182.214,235.946,-63.074,-177.424,7.058,148.565
C07981=1182.209,236.218,-63.102,-177.422,7.061,148.565
C07982=1182.204,236.489,-63.131,-177.418,7.064,148.564
C07983=1182.199,236.761,-63.159,-177.416,7.067,148.564
C07984=1182.194,237.033,-63.187,-177.413,7.069,148.564
C07985=1182.189,237.281,-63.214,-177.410,7.072,148.564
C07986=1182.185,237.530,-63.240,-177.408,7.074,148.564
C07987=1182.181,237.778,-63.266,-177.405,7.077,148.563
C07988=1182.176,238.027,-63.293,-177.402,7.078,148.563
C07989=1182.172,238.276,-63.318,-177.399,7.081,148.563
C07990=1182.168,238.524,-63.345,-177.397,7.083,148.563
C07991=1182.163,238.773,-63.371,-177.394,7.086,148.563
C07992=1182.158,239.021,-63.397,-177.392,7.088,148.563
C07993=1182.153,239.270,-63.424,-177.389,7.091,148.562
C07994=1182.149,239.518,-63.449,-177.386,7.093,148.562
C07995=1182.145,239.767,-63.476,-177.383,7.096,148.562
C07996=1182.140,240.016,-63.502,-177.381,7.098,148.562
C07997=1182.136,240.264,-63.529,-177.378,7.101,148.562
C07998=1182.131,240.513,-63.555,-177.376,7.103,148.561
C07999=1182.127,240.761,-63.582,-177.373,7.105,148.561
C08000=1182.123,241.010,-63.607,-177.370,7.107,148.561
C08001=1182.118,241.258,-63.634,-177.368,7.110,148.561
C08002=1182.114,241.507,-63.660,-177.365,7.113,148.561
C08003=1182.109,241.755,-63.687,-177.363,7.114,148.561
C08004=1182.105,242.004,-63.713,-177.360,7.117,148.560
C08005=1182.100,242.252,-63.740,-177.357,7.119,148.560
C08006=1182.096,242.501,-63.765,-177.355,7.122,148.560
C08007=1182.091,242.750,-63.792,-177.352,7.124,148.560
C08008=1182.087,242.999,-63.818,-177.349,7.127,148.560
C08009=1182.082,243.247,-63.845,-177.347,7.129,148.560
C08010=1182.079,243.495,-63.872,-177.344,7.132,148.559
C08011=1182.074,243.744,-63.898,-177.342,7.134,148.559
C08012=1182.070,243.993,-63.925,-177.339,7.137,148.559
C08013=1182.065,244.241,-63.952,-177.336,7.139,148.559
C08014=1182.061,244.490,-63.977,-177.334,7.142,148.559
C08015=1182.056,244.738,-64.004,-177.331,7.144,148.559
C08016=1182.051,244.987,-64.031,-177.328,7.146,148.558
C08017=1182.047,245.236,-64.057,-177.326,7.149,148.558
C08018=1182.043,245.484,-64.084,-177.323,7.151,148.558
C08019=1182.039,245.732,-64.111,-177.321,7.153,148.558
C08020=1182.034,245.981,-64.138,-177.318,7.156,148.558
C08021=1182.029,246.230,-64.164,-177.315,7.158,148.558
C08022=1182.025,246.478,-64.191,-177.312,7.161,148.557
C08023=1182.020,246.727,-64.218,-177.310,7.163,148.557
C08024=1182.017,246.975,-64.244,-177.307,7.166,148.557
C08025=1182.012,247.223,-64.271,-177.304,7.169,148.557
C08026=1182.007,247.472,-64.298,-177.302,7.171,148.557
C08027=1182.003,247.721,-64.324,-177.299,7.174,148.557
C08028=1181.998,247.969,-64.351,-177.297,7.176,148.557
C08029=1181.994,248.218,-64.378,-177.294,7.179,148.557
C08030=1181.990,248.466,-64.405,-177.291,7.181,148.556
C08031=1181.985,248.714,-64.432,-177.289,7.184,148.556
C08032=1181.980,248.963,-64.459,-177.287,7.186,148.556
C08033=1181.976,249.212,-64.485,-177.283,7.188,148.556
C08034=1181.972,249.460,-64.512,-177.281,7.191,148.556
C08035=1181.968,249.709,-64.539,-177.278,7.194,148.556
C08036=1181.963,249.958,-64.566,-177.276,7.195,148.555
C08037=1181.959,250.206,-64.593,-177.273,7.198,148.555
C08038=1181.954,250.454,-64.620,-177.270,7.201,148.555
C08039=1181.950,250.703,-64.647,-177.268,7.203,148.555
C08040=1181.945,250.951,-64.674,-177.265,7.206,148.555
C08041=1181.940,251.200,-64.701,-177.263,7.208,148.555
C08042=1181.936,251.448,-64.727,-177.260,7.211,148.555
C08043=1181.932,251.697,-64.754,-177.257,7.213,148.554
C08044=1181.928,251.946,-64.782,-177.255,7.216,148.554
C08045=1181.923,252.194,-64.809,-177.252,7.218,148.554
C08046=1181.918,252.443,-64.836,-177.249,7.221,148.554
C08047=1181.914,252.691,-64.862,-177.247,7.224,148.554
C08048=1181.910,252.939,-64.890,-177.244,7.226,148.554
C08049=1181.905,253.187,-64.917,-177.242,7.229,148.554
C08050=1181.901,253.436,-64.944,-177.239,7.231,148.553
C08051=1181.897,253.685,-64.972,-177.236,7.234,148.553
C08052=1181.892,253.934,-64.999,-177.234,7.236,148.553
C08053=1181.888,254.182,-65.025,-177.231,7.239,148.553
C08054=1181.884,254.430,-65.052,-177.228,7.242,148.553
C08055=1181.879,254.679,-65.079,-177.226,7.244,148.553
C08056=1181.875,254.927,-65.107,-177.223,7.247,148.553
C08057=1181.870,255.176,-65.134,-177.221,7.249,148.553
C08058=1181.866,255.424,-65.162,-177.218,7.251,148.552
C08059=1181.861,255.673,-65.189,-177.216,7.254,148.552
C08060=1181.857,255.921,-65.216,-177.213,7.257,148.552
C08061=1181.853,256.170,-65.244,-177.210,7.260,148.552
C08062=1181.848,256.418,-65.271,-177.208,7.261,148.552
C08063=1181.843,256.667,-65.298,-177.205,7.264,148.552
C08064=1181.839,256.915,-65.326,-177.203,7.267,148.552
C08065=1181.834,257.163,-65.353,-177.200,7.269,148.552
C08066=1181.831,257.412,-65.380,-177.197,7.272,148.551
C08067=1181.827,257.660,-65.407,-177.195,7.274,148.551
C08068=1181.822,257.908,-65.434,-177.192,7.277,148.551
C08069=1181.817,258.157,-65.462,-177.190,7.279,148.551
C08070=1181.814,258.406,-65.490,-177.186,7.282,148.551
C08071=1181.808,258.654,-65.517,-177.184,7.285,148.551
C08072=1181.804,258.903,-65.544,-177.182,7.287,148.551
C08073=1181.799,259.151,-65.572,-177.179,7.290,148.551
C08074=1181.795,259.400,-65.600,-177.177,7.292,148.551
C08075=1181.791,259.648,-65.627,-177.173,7.295,148.550
C08076=1181.786,259.896,-65.654,-177.171,7.298,148.550
C08077=1181.782,260.145,-65.683,-177.169,7.300,148.550
C08078=1181.778,260.393,-65.710,-177.166,7.303,148.550
C08079=1181.773,260.641,-65.737,-177.164,7.305,148.550
C08080=1181.769,260.890,-65.765,-177.160,7.308,148.550
C08081=1181.765,261.138,-65.793,-177.158,7.311,148.550
C08082=1181.760,261.387,-65.820,-177.156,7.313,148.550
C08083=1181.757,261.635,-65.848,-177.153,7.316,148.550
C08084=1181.752,261.884,-65.875,-177.150,7.319,148.550
C08085=1181.747,262.156,-65.905,-177.147,7.322,148.549
C08086=1181.742,262.430,-65.936,-177.144,7.325,148.549
C08087=1181.737,262.702,-65.966,-177.141,7.328,148.549
C08088=1181.732,262.976,-65.997,-177.138,7.330,148.549
C08089=1181.728,263.224,-66.025,-177.136,7.332,148.549
C08090=1181.724,263.473,-66.052,-177.133,7.335,148.549
C08091=1181.719,263.721,-66.080,-177.131,7.338,148.549
C08092=1181.715,263.970,-66.109,-177.128,7.341,148.549
C08093=1181.710,264.218,-66.136,-177.126,7.344,148.549
C08094=1181.706,264.466,-66.163,-177.123,7.345,148.548
C08095=1181.702,264.715,-66.192,-177.120,7.348,148.548
C08096=1181.697,264.963,-66.219,-177.118,7.351,148.548
C08097=1181.692,265.211,-66.247,-177.115,7.353,148.548
C08098=1181.689,265.460,-66.275,-177.113,7.356,148.548
C08099=1181.684,265.708,-66.302,-177.110,7.359,148.548
C08100=1181.680,265.957,-66.330,-177.107,7.361,148.548
C08101=1181.675,266.205,-66.359,-177.105,7.364,148.548
C08102=1181.671,266.453,-66.386,-177.102,7.367,148.548
C08103=1181.667,266.701,-66.415,-177.100,7.369,148.547
C08104=1181.662,266.950,-66.442,-177.097,7.372,148.547
C08105=1181.658,267.199,-66.470,-177.094,7.375,148.547
C08106=1181.654,267.447,-66.498,-177.092,7.378,148.547
C08107=1181.650,267.695,-66.526,-177.089,7.380,148.547
C08108=1181.645,267.944,-66.555,-177.086,7.383,148.547
C08109=1181.641,268.193,-66.582,-177.084,7.385,148.547
C08110=1181.636,268.441,-66.610,-177.081,7.388,148.547
C08111=1181.631,268.689,-66.638,-177.078,7.391,148.547
C08112=1181.627,268.937,-66.666,-177.076,7.393,148.547
C08113=1181.622,269.186,-66.695,-177.074,7.396,148.547
C08114=1181.619,269.434,-66.723,-177.071,7.399,148.547
C08115=1181.614,269.682,-66.751,-177.069,7.402,148.547
C08116=1181.610,269.931,-66.779,-177.065,7.404,148.546
C08117=1181.605,270.179,-66.807,-177.063,7.407,148.546
C08118=1181.601,270.428,-66.836,-177.061,7.409,148.546
C08119=1181.597,270.676,-66.864,-177.058,7.412,148.546
C08120=1181.593,270.924,-66.892,-177.055,7.415,148.546
C08121=1181.588,271.172,-66.920,-177.053,7.417,148.546
C08122=1181.584,271.421,-66.948,-177.050,7.420,148.546
C08123=1181.579,271.669,-66.977,-177.047,7.423,148.546
C08124=1181.575,271.918,-67.005,-177.045,7.426,148.546
C08125=1181.570,272.166,-67.033,-177.043,7.429,148.546
C08126=1181.566,272.414,-67.061,-177.039,7.431,148.546
C08127=1181.562,272.663,-67.090,-177.037,7.434,148.545
C08128=1181.558,272.911,-67.118,-177.034,7.436,148.545
C08129=1181.553,273.160,-67.147,-177.032,7.439,148.545
C08130=1181.549,273.408,-67.174,-177.029,7.442,148.545
C08131=1181.544,273.656,-67.204,-177.027,7.445,148.545
C08132=1181.540,273.904,-67.232,-177.024,7.447,148.545
C08133=1181.536,274.153,-67.260,-177.021,7.450,148.545
C08134=1181.532,274.402,-67.289,-177.019,7.453,148.545
C08135=1181.527,274.650,-67.317,-177.017,7.456,148.545
C08136=1181.523,274.898,-67.345,-177.014,7.459,148.545
C08137=1181.518,275.146,-67.374,-177.011,7.462,148.545
C08138=1181.515,275.394,-67.402,-177.009,7.464,148.545
C08139=1181.510,275.643,-67.431,-177.006,7.467,148.545
C08140=1181.505,275.891,-67.459,-177.003,7.470,148.545
C08141=1181.502,276.139,-67.488,-177.001,7.473,148.545
C08142=1181.496,276.388,-67.517,-176.999,7.475,148.545
C08143=1181.493,276.636,-67.545,-176.995,7.478,148.544
C08144=1181.488,276.884,-67.574,-176.993,7.481,148.544
C08145=1181.483,277.133,-67.603,-176.990,7.483,148.544
C08146=1181.480,277.381,-67.631,-176.988,7.486,148.544
C08147=1181.475,277.630,-67.660,-176.985,7.489,148.544
C08148=1181.470,277.878,-67.689,-176.982,7.492,148.544
C08149=1181.467,278.126,-67.717,-176.980,7.494,148.544
C08150=1181.462,278.375,-67.746,-176.977,7.497,148.544
C08151=1181.458,278.622,-67.774,-176.975,7.500,148.544
C08152=1181.454,278.871,-67.803,-176.972,7.503,148.544
C08153=1181.449,279.120,-67.832,-176.970,7.505,148.544
C08154=1181.444,279.368,-67.861,-176.967,7.508,148.544
C08155=1181.441,279.616,-67.889,-176.964,7.511,148.544
C08156=1181.436,279.865,-67.918,-176.962,7.514,148.544
C08157=1181.432,280.112,-67.947,-176.959,7.516,148.544
C08158=1181.428,280.361,-67.975,-176.957,7.519,148.544
C08159=1181.424,280.609,-68.005,-176.954,7.522,148.544
C08160=1181.419,280.858,-68.034,-176.951,7.525,148.544
C08161=1181.414,281.105,-68.063,-176.949,7.527,148.544
C08162=1181.411,281.354,-68.091,-176.946,7.530,148.543
C08163=1181.406,281.602,-68.120,-176.944,7.533,148.543
C08164=1181.401,281.850,-68.149,-176.941,7.536,148.543
C08165=1181.397,282.099,-68.178,-176.939,7.538,148.543
C08166=1181.393,282.347,-68.208,-176.936,7.541,148.543
C08167=1181.389,282.596,-68.236,-176.933,7.544,148.543
C08168=1181.385,282.843,-68.265,-176.931,7.547,148.543
C08169=1181.380,283.092,-68.293,-176.928,7.549,148.543
C08170=1181.376,283.340,-68.323,-176.926,7.552,148.543
C08171=1181.372,283.589,-68.352,-176.923,7.555,148.543
C08172=1181.367,283.837,-68.381,-176.920,7.558,148.543
C08173=1181.362,284.085,-68.410,-176.918,7.560,148.543
C08174=1181.359,284.333,-68.439,-176.915,7.563,148.543
C08175=1181.354,284.582,-68.468,-176.913,7.566,148.543
C08176=1181.350,284.830,-68.497,-176.910,7.569,148.543
C08177=1181.345,285.078,-68.526,-176.908,7.573,148.543
C08178=1181.341,285.326,-68.556,-176.905,7.575,148.543
C08179=1181.337,285.575,-68.585,-176.903,7.578,148.543
C08180=1181.333,285.823,-68.614,-176.900,7.581,148.543
C08181=1181.328,286.071,-68.643,-176.897,7.584,148.543
C08182=1181.324,286.319,-68.673,-176.895,7.586,148.543
C08183=1181.319,286.568,-68.701,-176.892,7.589,148.543
C08184=1181.315,286.816,-68.731,-176.890,7.592,148.543
C08185=1181.311,287.064,-68.760,-176.887,7.595,148.543
C08186=1181.307,287.313,-68.790,-176.884,7.598,148.543
C08187=1181.302,287.561,-68.819,-176.882,7.600,148.543
C08188=1181.298,287.809,-68.848,-176.879,7.603,148.543
C08189=1181.293,288.084,-68.880,-176.877,7.606,148.543
C08190=1181.289,288.359,-68.913,-176.873,7.610,148.543
C08191=1181.284,288.633,-68.945,-176.871,7.613,148.542
C08192=1181.279,288.908,-68.978,-176.868,7.616,148.542
C08193=1181.275,289.156,-69.007,-176.865,7.619,148.542
C08194=1181.270,289.404,-69.036,-176.862,7.622,148.542
C08195=1181.266,289.652,-69.066,-176.860,7.624,148.542
C08196=1181.262,289.900,-69.095,-176.857,7.627,148.542
C08197=1181.258,290.149,-69.125,-176.855,7.630,148.542
C08198=1181.253,290.397,-69.154,-176.852,7.633,148.542
C08199=1181.249,290.645,-69.184,-176.850,7.636,148.542
C08200=1181.245,290.894,-69.213,-176.848,7.639,148.542
C08201=1181.241,291.142,-69.242,-176.845,7.642,148.542
C08202=1181.237,291.390,-69.272,-176.842,7.644,148.542
C08203=1181.232,291.638,-69.301,-176.839,7.647,148.542
C08204=1181.228,291.887,-69.331,-176.837,7.650,148.542
C08205=1181.224,292.135,-69.362,-176.835,7.653,148.542
C08206=1181.219,292.382,-69.391,-176.832,7.656,148.542
C08207=1181.215,292.630,-69.420,-176.830,7.659,148.542
C08208=1181.211,292.879,-69.450,-176.827,7.662,148.542
C08209=1181.206,293.127,-69.479,-176.824,7.665,148.542
C08210=1181.201,293.375,-69.509,-176.822,7.667,148.542
C08211=1181.197,293.624,-69.539,-176.819,7.670,148.542
C08212=1181.193,293.871,-69.569,-176.816,7.673,148.542
C08213=1181.189,294.120,-69.598,-176.814,7.676,148.542
C08214=1181.185,294.368,-69.628,-176.811,7.679,148.542
C08215=1181.181,294.616,-69.657,-176.809,7.682,148.542
C08216=1181.176,294.865,-69.687,-176.807,7.685,148.542
C08217=1181.172,295.112,-69.717,-176.804,7.688,148.542
C08218=1181.168,295.361,-69.747,-176.801,7.690,148.542
C08219=1181.164,295.609,-69.776,-176.798,7.693,148.542
C08220=1181.159,295.857,-69.807,-176.796,7.696,148.542
C08221=1181.155,296.105,-69.836,-176.793,7.699,148.542
C08222=1181.151,296.353,-69.866,-176.791,7.702,148.542
C08223=1181.147,296.601,-69.896,-176.789,7.705,148.542
C08224=1181.142,296.850,-69.926,-176.786,7.708,148.542
C08225=1181.138,297.099,-69.956,-176.783,7.711,148.542
C08226=1181.134,297.346,-69.986,-176.780,7.714,148.542
C08227=1181.130,297.595,-70.016,-176.778,7.717,148.542
C08228=1181.125,297.843,-70.046,-176.776,7.719,148.542
C08229=1181.121,298.091,-70.076,-176.773,7.722,148.542
C08230=1181.117,298.339,-70.106,-176.771,7.725,148.542
C08231=1181.113,298.587,-70.136,-176.768,7.728,148.542
C08232=1181.109,298.835,-70.165,-176.765,7.731,148.542
C08233=1181.104,299.083,-70.196,-176.762,7.734,148.542
C08234=1181.100,299.332,-70.226,-176.760,7.738,148.542
C08235=1181.096,299.579,-70.256,-176.758,7.740,148.542
C08236=1181.091,299.828,-70.286,-176.755,7.743,148.542
C08237=1181.087,300.075,-70.316,-176.753,7.746,148.542
C08238=1181.083,300.325,-70.346,-176.750,7.749,148.542
C08239=1181.079,300.572,-70.377,-176.748,7.752,148.542
C08240=1181.075,300.821,-70.406,-176.745,7.755,148.542
C08241=1181.070,301.069,-70.437,-176.742,7.758,148.542
C08242=1181.066,301.317,-70.466,-176.740,7.760,148.542
C08243=1181.061,301.565,-70.497,-176.737,7.763,148.542
C08244=1181.057,301.813,-70.526,-176.735,7.767,148.542
C08245=1181.052,302.061,-70.557,-176.732,7.770,148.542
C08246=1181.049,302.309,-70.588,-176.729,7.773,148.542
C08247=1181.044,302.558,-70.618,-176.727,7.776,148.542
C08248=1181.040,302.806,-70.648,-176.724,7.779,148.542
C08249=1181.036,303.054,-70.679,-176.722,7.781,148.542
C08250=1181.032,303.302,-70.708,-176.720,7.784,148.542
C08251=1181.027,303.550,-70.739,-176.717,7.787,148.542
C08252=1181.024,303.798,-70.770,-176.714,7.790,148.542
C08253=1181.019,304.047,-70.800,-176.712,7.793,148.543
C08254=1181.015,304.294,-70.830,-176.709,7.796,148.543
C08255=1181.010,304.542,-70.860,-176.706,7.799,148.543
C08256=1181.006,304.790,-70.891,-176.704,7.802,148.543
C08257=1181.002,305.038,-70.921,-176.702,7.805,148.543
C08258=1180.998,305.287,-70.952,-176.699,7.808,148.543
C08259=1180.994,305.535,-70.982,-176.697,7.811,148.543
C08260=1180.989,305.783,-71.013,-176.694,7.814,148.543
C08261=1180.984,306.031,-71.044,-176.692,7.817,148.543
C08262=1180.981,306.280,-71.073,-176.689,7.820,148.543
C08263=1180.976,306.528,-71.104,-176.686,7.823,148.543
C08264=1180.972,306.775,-71.134,-176.683,7.826,148.543
C08265=1180.968,307.023,-71.165,-176.681,7.829,148.543
C08266=1180.963,307.271,-71.196,-176.679,7.832,148.543
C08267=1180.960,307.520,-71.226,-176.676,7.835,148.543
C08268=1180.955,307.768,-71.257,-176.674,7.838,148.543
C08269=1180.951,308.015,-71.288,-176.671,7.841,148.543
C08270=1180.947,308.264,-71.318,-176.669,7.844,148.543
C08271=1180.943,308.512,-71.349,-176.666,7.847,148.543
C08272=1180.938,308.760,-71.380,-176.664,7.850,148.543
C08273=1180.934,309.007,-71.410,-176.661,7.853,148.543
C08274=1180.930,309.256,-71.441,-176.658,7.856,148.543
C08275=1180.926,309.504,-71.472,-176.657,7.859,148.543
C08276=1180.921,309.752,-71.503,-176.654,7.862,148.543
C08277=1180.918,310.000,-71.533,-176.651,7.865,148.543
C08278=1180.913,310.248,-71.564,-176.649,7.868,148.543
C08279=1180.908,310.496,-71.595,-176.646,7.871,148.543
C08280=1180.904,310.744,-71.626,-176.643,7.874,148.543
C08281=1180.901,310.993,-71.656,-176.641,7.877,148.544
C08282=1180.896,311.240,-71.687,-176.638,7.880,148.544
C08283=1180.891,311.488,-71.718,-176.636,7.883,148.544
C08284=1180.887,311.737,-71.749,-176.633,7.886,148.544
C08285=1180.883,311.985,-71.780,-176.631,7.889,148.544
C08286=1180.879,312.233,-71.810,-176.629,7.892,148.544
C08287=1180.875,312.481,-71.842,-176.626,7.895,148.544
C08288=1180.871,312.729,-71.872,-176.624,7.898,148.544
C08289=1180.867,312.977,-71.903,-176.621,7.901,148.544
C08290=1180.862,313.225,-71.934,-176.619,7.904,148.544
C08291=1180.857,313.473,-71.965,-176.616,7.907,148.544
C08292=1180.854,313.721,-71.996,-176.613,7.910,148.544
C08293=1180.849,313.998,-72.031,-176.611,7.914,148.544
C08294=1180.844,314.274,-72.065,-176.608,7.917,148.544
C08295=1180.839,314.551,-72.100,-176.605,7.920,148.544
C08296=1180.835,314.828,-72.134,-176.602,7.923,148.544
C08297=1180.831,315.076,-72.166,-176.600,7.927,148.544
C08298=1180.827,315.324,-72.197,-176.597,7.930,148.544
C08299=1180.822,315.572,-72.228,-176.595,7.933,148.545
C08300=1180.818,315.820,-72.259,-176.592,7.936,148.545
C08301=1180.814,316.068,-72.290,-176.589,7.939,148.545
C08302=1180.810,316.317,-72.321,-176.587,7.942,148.545
C08303=1180.805,316.564,-72.353,-176.584,7.945,148.545
C08304=1180.801,316.812,-72.384,-176.582,7.949,148.545
C08305=1180.798,317.060,-72.415,-176.579,7.952,148.545
C08306=1180.793,317.308,-72.446,-176.577,7.955,148.545
C08307=1180.789,317.556,-72.477,-176.574,7.958,148.545
C08308=1180.785,317.804,-72.508,-176.572,7.961,148.545
C08309=1180.781,318.052,-72.539,-176.570,7.963,148.545
C08310=1180.777,318.300,-72.571,-176.567,7.966,148.545
C08311=1180.773,318.548,-72.602,-176.565,7.969,148.545
C08312=1180.768,318.796,-72.633,-176.562,7.973,148.546
C08313=1180.763,319.045,-72.665,-176.560,7.976,148.546
C08314=1180.759,319.292,-72.697,-176.557,7.979,148.546
C08315=1180.755,319.540,-72.728,-176.555,7.982,148.546
C08316=1180.751,319.788,-72.759,-176.552,7.985,148.546
C08317=1180.747,320.036,-72.791,-176.550,7.988,148.546
C08318=1180.743,320.284,-72.822,-176.547,7.991,148.546
C08319=1180.739,320.532,-72.854,-176.545,7.995,148.546
C08320=1180.734,320.780,-72.884,-176.542,7.998,148.546
C08321=1180.730,321.028,-72.916,-176.540,8.001,148.546
C08322=1180.726,321.275,-72.948,-176.537,8.004,148.546
C08323=1180.722,321.524,-72.979,-176.535,8.007,148.546
C08324=1180.718,321.771,-73.010,-176.532,8.010,148.546
C08325=1180.713,322.020,-73.043,-176.530,8.014,148.547
C08326=1180.709,322.268,-73.074,-176.527,8.017,148.547
C08327=1180.705,322.516,-73.105,-176.525,8.020,148.547
C08328=1180.701,322.764,-73.137,-176.523,8.022,148.547
C08329=1180.697,323.012,-73.168,-176.520,8.025,148.547
C08330=1180.693,323.260,-73.200,-176.518,8.028,148.547
C08331=1180.689,323.507,-73.231,-176.515,8.032,148.547
C08332=1180.684,323.756,-73.264,-176.513,8.035,148.547
C08333=1180.681,324.004,-73.296,-176.510,8.038,148.547
C08334=1180.676,324.252,-73.326,-176.508,8.041,148.547
C08335=1180.672,324.500,-73.358,-176.505,8.044,148.548
C08336=1180.668,324.748,-73.391,-176.503,8.047,148.548
C08337=1180.664,324.995,-73.422,-176.500,8.051,148.548
C08338=1180.660,325.243,-73.454,-176.498,8.054,148.548
C08339=1180.656,325.491,-73.485,-176.495,8.057,148.548
C08340=1180.652,325.739,-73.517,-176.493,8.060,148.548
C08341=1180.647,325.988,-73.549,-176.491,8.063,148.548
C08342=1180.643,326.235,-73.581,-176.488,8.066,148.548
C08343=1180.639,326.483,-73.612,-176.486,8.070,148.548
C08344=1180.635,326.731,-73.645,-176.483,8.073,148.549
C08345=1180.630,326.979,-73.676,-176.481,8.076,148.549
C08346=1180.627,327.227,-73.708,-176.478,8.079,148.549
C08347=1180.622,327.475,-73.741,-176.476,8.082,148.549
C08348=1180.618,327.722,-73.772,-176.473,8.085,148.549
C08349=1180.614,327.970,-73.804,-176.471,8.088,148.549
C08350=1180.610,328.219,-73.836,-176.468,8.092,148.549
C08351=1180.605,328.466,-73.868,-176.466,8.095,148.549
C08352=1180.602,328.714,-73.900,-176.463,8.098,148.549
C08353=1180.597,328.963,-73.932,-176.461,8.101,148.550
C08354=1180.593,329.210,-73.964,-176.458,8.104,148.550
C08355=1180.589,329.458,-73.995,-176.456,8.108,148.550
C08356=1180.585,329.706,-74.028,-176.454,8.111,148.550
C08357=1180.580,329.954,-74.059,-176.451,8.114,148.550
C08358=1180.576,330.202,-74.092,-176.449,8.117,148.550
C08359=1180.572,330.450,-74.124,-176.446,8.120,148.550
C08360=1180.568,330.698,-74.157,-176.444,8.124,148.550
C08361=1180.564,330.945,-74.188,-176.442,8.127,148.551
C08362=1180.560,331.193,-74.220,-176.439,8.130,148.551
C08363=1180.556,331.441,-74.253,-176.437,8.133,148.551
C08364=1180.552,331.689,-74.284,-176.435,8.136,148.551
C08365=1180.547,331.937,-74.317,-176.432,8.139,148.551
C08366=1180.544,332.185,-74.349,-176.430,8.142,148.551
C08367=1180.539,332.433,-74.382,-176.428,8.145,148.551
C08368=1180.535,332.681,-74.413,-176.425,8.148,148.551
C08369=1180.530,332.929,-74.445,-176.423,8.152,148.552
C08370=1180.527,333.176,-74.478,-176.420,8.155,148.552
C08371=1180.523,333.424,-74.510,-176.418,8.158,148.552
C08372=1180.519,333.672,-74.542,-176.415,8.161,148.552
C08373=1180.514,333.920,-74.574,-176.413,8.165,148.552
C08374=1180.510,334.167,-74.607,-176.410,8.168,148.552
C08375=1180.506,334.416,-74.639,-176.408,8.171,148.553
C08376=1180.502,334.664,-74.672,-176.406,8.174,148.553
C08377=1180.498,334.912,-74.704,-176.404,8.178,148.553
C08378=1180.493,335.159,-74.736,-176.401,8.181,148.553
C08379=1180.490,335.407,-74.769,-176.399,8.184,148.553
C08380=1180.485,335.655,-74.801,-176.396,8.187,148.553
C08381=1180.481,335.903,-74.834,-176.394,8.190,148.554
C08382=1180.477,336.151,-74.866,-176.391,8.193,148.554
C08383=1180.473,336.399,-74.899,-176.389,8.198,148.554
C08384=1180.470,336.647,-74.931,-176.386,8.201,148.554
C08385=1180.464,336.894,-74.963,-176.384,8.204,148.554
C08386=1180.460,337.142,-74.997,-176.381,8.207,148.554
C08387=1180.457,337.390,-75.028,-176.379,8.211,148.554
C08388=1180.452,337.638,-75.062,-176.377,8.214,148.555
C08389=1180.448,337.886,-75.094,-176.375,8.217,148.555
C08390=1180.445,338.133,-75.127,-176.372,8.220,148.555
C08391=1180.440,338.382,-75.159,-176.370,8.223,148.555
C08392=1180.435,338.629,-75.192,-176.367,8.227,148.555
C08393=1180.432,338.877,-75.224,-176.365,8.230,148.556
C08394=1180.428,339.125,-75.257,-176.363,8.233,148.556
C08395=1180.423,339.372,-75.290,-176.361,8.237,148.556
C08396=1180.419,339.621,-75.322,-176.358,8.240,148.556
C08397=1180.415,339.899,-75.359,-176.356,8.243,148.556
C08398=1180.411,340.178,-75.396,-176.353,8.247,148.556
C08399=1180.406,340.457,-75.433,-176.351,8.250,148.557
C08400=1180.401,340.736,-75.470,-176.348,8.255,148.557
C08401=1180.397,340.984,-75.502,-176.345,8.258,148.557
C08402=1180.392,341.232,-75.535,-176.343,8.261,148.557
C08403=1180.388,341.480,-75.568,-176.340,8.264,148.557
C08404=1180.384,341.728,-75.601,-176.338,8.268,148.558
C08405=1180.381,341.975,-75.633,-176.336,8.271,148.558
C08406=1180.376,342.223,-75.667,-176.334,8.274,148.558
C08407=1180.372,342.471,-75.700,-176.331,8.278,148.558
C08408=1180.368,342.719,-75.732,-176.329,8.281,148.558
C08409=1180.364,342.967,-75.765,-176.327,8.284,148.559
C08410=1180.360,343.215,-75.799,-176.325,8.287,148.559
C08411=1180.356,343.462,-75.831,-176.322,8.290,148.559
C08412=1180.352,343.711,-75.864,-176.320,8.294,148.559
C08413=1180.348,343.958,-75.897,-176.317,8.297,148.559
C08414=1180.343,344.206,-75.930,-176.315,8.300,148.560
C08415=1180.339,344.454,-75.963,-176.313,8.304,148.560
C08416=1180.335,344.701,-75.996,-176.311,8.307,148.560
C08417=1180.331,344.949,-76.029,-176.308,8.310,148.560
C08418=1180.327,345.197,-76.062,-176.306,8.314,148.560
C08419=1180.323,345.445,-76.096,-176.303,8.318,148.561
C08420=1180.319,345.692,-76.129,-176.301,8.321,148.561
C08421=1180.314,345.941,-76.161,-176.299,8.324,148.561
C08422=1180.310,346.188,-76.194,-176.296,8.328,148.561
C08423=1180.306,346.436,-76.228,-176.294,8.331,148.562
C08424=1180.302,346.684,-76.261,-176.292,8.334,148.562
C08425=1180.298,346.931,-76.293,-176.290,8.338,148.562
C08426=1180.294,347.179,-76.326,-176.287,8.341,148.562
C08427=1180.290,347.427,-76.360,-176.285,8.344,148.562
C08428=1180.286,347.675,-76.393,-176.283,8.348,148.563
C08429=1180.282,347.922,-76.426,-176.281,8.351,148.563
C08430=1180.277,348.170,-76.460,-176.278,8.354,148.563
C08431=1180.273,348.417,-76.493,-176.276,8.358,148.563
C08432=1180.269,348.665,-76.527,-176.274,8.361,148.564
C08433=1180.265,348.914,-76.560,-176.272,8.364,148.564
C08434=1180.261,349.161,-76.593,-176.270,8.368,148.564
C08435=1180.257,349.409,-76.626,-176.267,8.371,148.564
C08436=1180.253,349.657,-76.660,-176.265,8.374,148.565
C08437=1180.249,349.904,-76.693,-176.262,8.379,148.565
C08438=1180.245,350.152,-76.726,-176.260,8.382,148.565
C08439=1180.241,350.399,-76.760,-176.258,8.385,148.565
C08440=1180.237,350.647,-76.793,-176.256,8.389,148.566
C08441=1180.233,350.895,-76.826,-176.254,8.392,148.566
C08442=1180.229,351.143,-76.860,-176.251,8.395,148.566
C08443=1180.224,351.391,-76.894,-176.249,8.399,148.566
C08444=1180.220,351.638,-76.927,-176.247,8.402,148.567
C08445=1180.216,351.886,-76.960,-176.245,8.405,148.567
C08446=1180.212,352.134,-76.994,-176.243,8.409,148.567
C08447=1180.208,352.381,-77.027,-176.241,8.412,148.567
C08448=1180.204,352.629,-77.061,-176.238,8.416,148.568
C08449=1180.201,352.877,-77.094,-176.236,8.419,148.568
C08450=1180.196,353.125,-77.128,-176.234,8.422,148.568
C08451=1180.192,353.372,-77.162,-176.231,8.427,148.569
C08452=1180.188,353.620,-77.195,-176.229,8.430,148.569
C08453=1180.184,353.867,-77.229,-176.227,8.433,148.569
C08454=1180.180,354.115,-77.262,-176.225,8.437,148.569
C08455=1180.175,354.364,-77.296,-176.223,8.440,148.570
C08456=1180.172,354.611,-77.330,-176.221,8.444,148.570
C08457=1180.167,354.858,-77.363,-176.218,8.447,148.570
C08458=1180.164,355.105,-77.397,-176.216,8.450,148.571
C08459=1180.159,355.354,-77.431,-176.214,8.454,148.571
C08460=1180.155,355.602,-77.464,-176.212,8.457,148.571
C08461=1180.151,355.849,-77.498,-176.210,8.461,148.571
C08462=1180.147,356.097,-77.531,-176.208,8.464,148.572
C08463=1180.143,356.345,-77.566,-176.205,8.468,148.572
C08464=1180.139,356.593,-77.599,-176.203,8.472,148.572
C08465=1180.135,356.840,-77.633,-176.201,8.475,148.573
C08466=1180.130,357.088,-77.667,-176.199,8.478,148.573
C08467=1180.127,357.336,-77.701,-176.197,8.482,148.573
C08468=1180.123,357.583,-77.735,-176.195,8.485,148.573
C08469=1180.119,357.830,-77.768,-176.192,8.489,148.574
C08470=1180.115,358.078,-77.803,-176.190,8.492,148.574
C08471=1180.111,358.326,-77.836,-176.188,8.496,148.574
C08472=1180.107,358.573,-77.870,-176.186,8.499,148.575
C08473=1180.103,358.821,-77.904,-176.184,8.502,148.575
C08474=1180.099,359.069,-77.938,-176.182,8.507,148.575
C08475=1180.095,359.317,-77.972,-176.179,8.510,148.576
C08476=1180.090,359.564,-78.006,-176.178,8.514,148.576
C08477=1180.087,359.811,-78.039,-176.175,8.517,148.576
C08478=1180.083,360.060,-78.074,-176.174,8.521,148.577
C08479=1180.079,360.307,-78.108,-176.171,8.524,148.577
C08480=1180.074,360.555,-78.142,-176.169,8.528,148.577
C08481=1180.071,360.803,-78.176,-176.167,8.531,148.578
C08482=1180.067,361.050,-78.210,-176.165,8.535,148.578
C08483=1180.062,361.297,-78.245,-176.164,8.538,148.578
C08484=1180.059,361.546,-78.278,-176.161,8.542,148.579
C08485=1180.054,361.793,-78.312,-176.159,8.545,148.579
C08486=1180.050,362.040,-78.346,-176.158,8.549,148.580
C08487=1180.046,362.288,-78.381,-176.155,8.552,148.580
C08488=1180.042,362.536,-78.414,-176.154,8.556,148.580
C08489=1180.038,362.784,-78.449,-176.152,8.559,148.581
C08490=1180.035,363.031,-78.483,-176.149,8.563,148.581
C08491=1180.030,363.279,-78.518,-176.148,8.566,148.581
C08492=1180.027,363.526,-78.552,-176.146,8.570,148.582
C08493=1180.022,363.774,-78.586,-176.144,8.574,148.582
C08494=1180.019,364.022,-78.620,-176.142,8.577,148.583
C08495=1180.014,364.269,-78.655,-176.140,8.580,148.583
C08496=1180.010,364.517,-78.688,-176.138,8.584,148.583
C08497=1180.006,364.765,-78.723,-176.136,8.588,148.584
C08498=1180.002,365.012,-78.757,-176.134,8.591,148.584
C08499=1179.998,365.260,-78.792,-176.133,8.595,148.585
C08500=1179.995,365.507,-78.825,-176.131,8.599,148.585
C08501=1179.990,365.789,-78.865,-176.129,8.602,148.585
C08502=1179.986,366.070,-78.904,-176.127,8.607,148.586
C08503=1179.981,366.352,-78.943,-176.125,8.610,148.586
C08504=1179.976,366.633,-78.983,-176.122,8.615,148.587
C08505=1179.973,366.881,-79.017,-176.121,8.618,148.587
C08506=1179.968,367.129,-79.051,-176.119,8.622,148.588
C08507=1179.965,367.376,-79.086,-176.117,8.625,148.588
C08508=1179.960,367.624,-79.120,-176.116,8.628,148.588
C08509=1179.956,367.871,-79.155,-176.114,8.632,148.589
C08510=1179.952,368.119,-79.189,-176.112,8.636,148.590
C08511=1179.948,368.367,-79.223,-176.111,8.639,148.590
C08512=1179.944,368.615,-79.258,-176.109,8.643,148.590
C08513=1179.940,368.862,-79.292,-176.107,8.647,148.591
C08514=1179.936,369.110,-79.327,-176.106,8.649,148.591
C08515=1179.932,369.357,-79.362,-176.104,8.653,148.592
C08516=1179.929,369.605,-79.396,-176.103,8.657,148.592
C08517=1179.924,369.852,-79.431,-176.101,8.661,148.593
C08518=1179.920,370.100,-79.466,-176.099,8.664,148.593
C08519=1179.915,370.347,-79.500,-176.097,8.668,148.594
C08520=1179.912,370.595,-79.534,-176.096,8.671,148.594
C08521=1179.908,370.842,-79.569,-176.094,8.675,148.595
C08522=1179.904,371.090,-79.604,-176.093,8.678,148.595
C08523=1179.900,371.337,-79.638,-176.091,8.682,148.596
C08524=1179.896,371.585,-79.673,-176.090,8.685,148.596
C08525=1179.892,371.832,-79.708,-176.088,8.689,148.596
C08526=1179.888,372.080,-79.743,-176.087,8.692,148.597
C08527=1179.883,372.328,-79.777,-176.085,8.695,148.597
C08528=1179.880,372.576,-79.812,-176.084,8.699,148.598
C08529=1179.876,372.822,-79.847,-176.082,8.703,148.599
C08530=1179.872,373.070,-79.882,-176.081,8.706,148.599
C08531=1179.868,373.319,-79.917,-176.080,8.709,148.600
C08532=1179.864,373.565,-79.951,-176.078,8.713,148.600
C08533=1179.860,373.813,-79.986,-176.077,8.716,148.601
C08534=1179.856,374.061,-80.020,-176.076,8.720,148.601
C08535=1179.852,374.308,-80.056,-176.074,8.724,148.602
C08536=1179.848,374.556,-80.090,-176.073,8.727,148.602
C08537=1179.844,374.803,-80.126,-176.072,8.731,148.603
C08538=1179.841,375.051,-80.160,-176.070,8.734,148.603
C08539=1179.836,375.298,-80.195,-176.069,8.737,148.604
C08540=1179.833,375.546,-80.230,-176.067,8.741,148.604
C08541=1179.828,375.793,-80.265,-176.066,8.744,148.605
C08542=1179.824,376.041,-80.300,-176.065,8.748,148.606
C08543=1179.820,376.288,-80.335,-176.064,8.751,148.606
C08544=1179.816,376.536,-80.370,-176.062,8.755,148.607
C08545=1179.813,376.783,-80.404,-176.061,8.758,148.607
C08546=1179.809,377.030,-80.440,-176.060,8.762,148.608
C08547=1179.805,377.278,-80.475,-176.059,8.765,148.608
C08548=1179.800,377.525,-80.510,-176.058,8.768,148.609
C08549=1179.796,377.773,-80.545,-176.057,8.772,148.609
C08550=1179.793,378.021,-80.580,-176.056,8.775,148.610
C08551=1179.788,378.268,-80.615,-176.054,8.779,148.611
C08552=1179.785,378.516,-80.650,-176.054,8.782,148.611
C08553=1179.781,378.764,-80.685,-176.053,8.785,148.612
C08554=1179.776,379.011,-80.720,-176.051,8.789,148.612
C08555=1179.772,379.259,-80.755,-176.050,8.792,148.613
C08556=1179.768,379.506,-80.790,-176.050,8.795,148.614
C08557=1179.764,379.754,-80.825,-176.048,8.799,148.614
C08558=1179.760,380.001,-80.860,-176.047,8.802,148.615
C08559=1179.756,380.248,-80.896,-176.046,8.805,148.615
C08560=1179.752,380.496,-80.931,-176.045,8.809,148.616
C08561=1179.749,380.744,-80.966,-176.044,8.812,148.616
C08562=1179.744,380.990,-81.001,-176.044,8.815,148.617
C08563=1179.740,381.239,-81.036,-176.043,8.818,148.618
C08564=1179.737,381.486,-81.072,-176.042,8.821,148.618
C08565=1179.732,381.733,-81.106,-176.041,8.825,148.619
C08566=1179.728,381.981,-81.142,-176.040,8.828,148.619
C08567=1179.725,382.228,-81.177,-176.039,8.831,148.620
C08568=1179.720,382.476,-81.212,-176.038,8.835,148.621
C08569=1179.716,382.723,-81.247,-176.037,8.838,148.621
C08570=1179.713,382.971,-81.283,-176.036,8.841,148.622
C08571=1179.709,383.218,-81.318,-176.036,8.844,148.623
C08572=1179.705,383.466,-81.353,-176.035,8.847,148.623
C08573=1179.701,383.713,-81.388,-176.034,8.850,148.624
C08574=1179.697,383.960,-81.423,-176.034,8.853,148.624
C08575=1179.693,384.208,-81.458,-176.033,8.856,148.625
C08576=1179.689,384.456,-81.494,-176.032,8.860,148.626
C08577=1179.685,384.703,-81.529,-176.032,8.863,148.626
C08578=1179.681,384.950,-81.565,-176.031,8.866,148.627
C08579=1179.677,385.197,-81.600,-176.030,8.869,148.628
C08580=1179.673,385.446,-81.635,-176.029,8.873,148.628
C08581=1179.669,385.692,-81.670,-176.029,8.876,148.629
C08582=1179.666,385.940,-81.706,-176.028,8.879,148.629
C08583=1179.662,386.187,-81.741,-176.027,8.882,148.630
C08584=1179.657,386.436,-81.777,-176.027,8.885,148.631
C08585=1179.653,386.683,-81.812,-176.027,8.888,148.631
C08586=1179.649,386.930,-81.847,-176.026,8.891,148.632
C08587=1179.646,387.178,-81.883,-176.025,8.894,148.633
C08588=1179.641,387.424,-81.918,-176.025,8.897,148.633
C08589=1179.638,387.672,-81.954,-176.025,8.900,148.634
C08590=1179.634,387.919,-81.989,-176.024,8.903,148.635
C08591=1179.630,388.168,-82.024,-176.023,8.906,148.635
C08592=1179.625,388.415,-82.060,-176.023,8.910,148.636
C08593=1179.621,388.662,-82.095,-176.023,8.912,148.637
C08594=1179.618,388.910,-82.131,-176.022,8.915,148.637
C08595=1179.614,389.157,-82.166,-176.022,8.917,148.638
C08596=1179.610,389.404,-82.202,-176.022,8.921,148.639
C08597=1179.606,389.651,-82.237,-176.021,8.924,148.639
C08598=1179.602,389.899,-82.273,-176.021,8.926,148.640
C08599=1179.598,390.147,-82.308,-176.020,8.930,148.641
C08600=1179.594,390.395,-82.344,-176.020,8.932,148.641
C08601=1179.590,390.642,-82.379,-176.019,8.935,148.642
C08602=1179.586,390.889,-82.414,-176.020,8.938,148.643
C08603=1179.582,391.137,-82.450,-176.019,8.941,148.643
C08604=1179.579,391.384,-82.486,-176.019,8.943,148.644
C08605=1179.574,391.668,-82.527,-176.019,8.947,148.645
C08606=1179.570,391.953,-82.567,-176.018,8.950,148.645
C08607=1179.565,392.236,-82.608,-176.018,8.954,148.646
C08608=1179.560,392.521,-82.649,-176.018,8.956,148.647
C08609=1179.557,392.769,-82.685,-176.017,8.959,148.647
C08610=1179.552,393.015,-82.720,-176.017,8.962,148.648
C08611=1179.549,393.263,-82.755,-176.017,8.964,148.649
C08612=1179.544,393.511,-82.792,-176.017,8.968,148.650
C08613=1179.541,393.758,-82.827,-176.017,8.970,148.650
C08614=1179.537,394.006,-82.863,-176.017,8.972,148.651
C08615=1179.533,394.252,-82.898,-176.016,8.976,148.652
C08616=1179.529,394.500,-82.933,-176.016,8.978,148.652
C08617=1179.525,394.748,-82.970,-176.016,8.981,148.653
C08618=1179.521,394.995,-83.005,-176.016,8.983,148.654
C08619=1179.517,395.243,-83.041,-176.015,8.986,148.654
C08620=1179.513,395.490,-83.076,-176.016,8.989,148.655
C08621=1179.509,395.737,-83.112,-176.015,8.991,148.655
C08622=1179.505,395.985,-83.148,-176.016,8.994,148.656
C08623=1179.501,396.232,-83.183,-176.016,8.996,148.657
C08624=1179.498,396.480,-83.219,-176.015,8.998,148.657
C08625=1179.493,396.727,-83.254,-176.016,9.001,148.658
C08626=1179.489,396.974,-83.291,-176.015,9.004,148.659
C08627=1179.486,397.221,-83.326,-176.015,9.007,148.659
C08628=1179.482,397.469,-83.362,-176.015,9.009,148.660
C08629=1179.478,397.717,-83.398,-176.015,9.012,148.661
C08630=1179.473,397.963,-83.433,-176.015,9.014,148.661
C08631=1179.470,398.211,-83.469,-176.015,9.016,148.662
C08632=1179.465,398.459,-83.505,-176.015,9.019,148.662
C08633=1179.462,398.706,-83.540,-176.015,9.022,148.663
C08634=1179.458,398.954,-83.576,-176.015,9.024,148.664
C08635=1179.454,399.201,-83.611,-176.015,9.026,148.664
C08636=1179.449,399.448,-83.647,-176.015,9.029,148.665
C08637=1179.446,399.695,-83.683,-176.015,9.031,148.666
C08638=1179.442,399.943,-83.719,-176.015,9.034,148.666
C08639=1179.438,400.191,-83.755,-176.015,9.036,148.667
C08640=1179.434,400.438,-83.791,-176.015,9.039,148.668
C08641=1179.430,400.686,-83.826,-176.015,9.041,148.668
C08642=1179.425,400.933,-83.862,-176.015,9.043,148.669
C08643=1179.422,401.180,-83.898,-176.015,9.046,148.669
C08644=1179.418,401.428,-83.933,-176.015,9.047,148.670
C08645=1179.415,401.675,-83.969,-176.015,9.050,148.671
C08646=1179.410,401.922,-84.006,-176.015,9.052,148.671
C08647=1179.407,402.170,-84.041,-176.015,9.055,148.672
C08648=1179.403,402.417,-84.077,-176.015,9.057,148.673
C08649=1179.398,402.664,-84.112,-176.015,9.060,148.673
C08650=1179.394,402.912,-84.148,-176.015,9.062,148.674
C08651=1179.391,403.159,-84.184,-176.016,9.064,148.674
C08652=1179.387,403.407,-84.220,-176.015,9.066,148.675
C08653=1179.383,403.654,-84.256,-176.016,9.068,148.676
C08654=1179.379,403.902,-84.291,-176.015,9.071,148.676
C08655=1179.375,404.149,-84.328,-176.016,9.073,148.677
C08656=1179.371,404.396,-84.363,-176.016,9.075,148.677
C08657=1179.367,404.643,-84.399,-176.016,9.077,148.678
C08658=1179.363,404.891,-84.435,-176.016,9.080,148.679
C08659=1179.359,405.138,-84.471,-176.016,9.082,148.679
C08660=1179.356,405.386,-84.506,-176.016,9.084,148.680
C08661=1179.351,405.633,-84.543,-176.016,9.086,148.681
C08662=1179.348,405.881,-84.579,-176.016,9.088,148.681
C08663=1179.344,406.127,-84.614,-176.017,9.090,148.682
C08664=1179.339,406.375,-84.650,-176.017,9.092,148.682
C08665=1179.336,406.623,-84.686,-176.017,9.095,148.683
C08666=1179.332,406.870,-84.722,-176.017,9.096,148.683
C08667=1179.328,407.117,-84.758,-176.017,9.099,148.684
C08668=1179.324,407.365,-84.794,-176.017,9.101,148.685
C08669=1179.320,407.613,-84.830,-176.017,9.103,148.685
C08670=1179.316,407.860,-84.866,-176.017,9.105,148.686
C08671=1179.312,408.106,-84.901,-176.017,9.108,148.686
C08672=1179.308,408.354,-84.937,-176.018,9.109,148.687
C08673=1179.304,408.602,-84.973,-176.018,9.112,148.687
C08674=1179.301,408.849,-85.009,-176.018,9.114,148.688
C08675=1179.296,409.096,-85.045,-176.018,9.116,148.689
C08676=1179.293,409.344,-85.081,-176.018,9.118,148.689
C08677=1179.288,409.591,-85.118,-176.019,9.120,148.690
C08678=1179.285,409.839,-85.153,-176.018,9.122,148.690
C08679=1179.281,410.086,-85.189,-176.018,9.124,148.691
C08680=1179.277,410.334,-85.225,-176.019,9.126,148.692
C08681=1179.273,410.580,-85.261,-176.018,9.128,148.692
C08682=1179.269,410.828,-85.296,-176.019,9.130,148.693
C08683=1179.265,411.075,-85.332,-176.019,9.132,148.693
C08684=1179.261,411.322,-85.369,-176.019,9.134,148.694
C08685=1179.257,411.570,-85.405,-176.019,9.136,148.694
C08686=1179.253,411.818,-85.440,-176.020,9.138,148.695
C08687=1179.249,412.065,-85.477,-176.019,9.140,148.695
C08688=1179.246,412.312,-85.513,-176.019,9.142,148.696
C08689=1179.242,412.560,-85.548,-176.019,9.143,148.696
C08690=1179.238,412.808,-85.584,-176.020,9.146,148.697
C08691=1179.234,413.054,-85.620,-176.020,9.147,148.698
C08692=1179.229,413.302,-85.657,-176.020,9.150,148.698
C08693=1179.225,413.549,-85.692,-176.020,9.151,148.699
C08694=1179.222,413.796,-85.728,-176.020,9.154,148.699
C08695=1179.218,414.044,-85.764,-176.020,9.155,148.700
C08696=1179.214,414.291,-85.800,-176.020,9.157,148.700
C08697=1179.210,414.539,-85.837,-176.020,9.159,148.701
C08698=1179.206,414.786,-85.872,-176.021,9.161,148.701
C08699=1179.202,415.034,-85.909,-176.021,9.163,148.702
C08700=1179.199,415.281,-85.945,-176.021,9.164,148.702
C08701=1179.194,415.514,-85.978,-176.021,9.167,148.703
C08702=1179.191,415.747,-86.012,-176.021,9.168,148.703
C08703=1179.188,415.981,-86.046,-176.021,9.170,148.704
C08704=1179.188,416.214,-86.080,-176.021,9.172,148.704
C08705=1179.187,416.447,-86.113,-176.021,9.173,148.705
C08706=1179.187,416.680,-86.147,-176.021,9.175,148.705
C08707=1179.189,416.912,-86.180,-176.021,9.177,148.706
C08708=1179.191,417.145,-86.213,-176.021,9.178,148.706
C08709=1178.771,417.146,-86.257,-176.025,9.189,148.710
C08710=1178.768,416.912,-86.223,-176.024,9.188,148.709
C08711=1178.766,416.678,-86.189,-176.024,9.186,148.709
C08712=1178.765,416.443,-86.156,-176.024,9.184,148.708
C08713=1178.766,416.209,-86.122,-176.024,9.182,148.708
C08714=1178.768,415.974,-86.088,-176.024,9.181,148.708
C08715=1178.769,415.739,-86.054,-176.025,9.179,148.707
C08716=1178.774,415.505,-86.019,-176.024,9.177,148.706
C08717=1178.777,415.269,-85.985,-176.023,9.176,148.706
C08718=1178.780,415.022,-85.949,-176.024,9.174,148.705
C08719=1178.785,414.775,-85.914,-176.023,9.172,148.705
C08720=1178.789,414.528,-85.877,-176.024,9.170,148.704
C08721=1178.793,414.280,-85.841,-176.023,9.168,148.704
C08722=1178.797,414.033,-85.806,-176.023,9.166,148.703
C08723=1178.800,413.786,-85.769,-176.023,9.164,148.703
C08724=1178.805,413.538,-85.733,-176.023,9.162,148.702
C08725=1178.808,413.290,-85.698,-176.023,9.161,148.702
C08726=1178.812,413.043,-85.661,-176.023,9.158,148.701
C08727=1178.816,412.796,-85.625,-176.023,9.157,148.701
C08728=1178.820,412.548,-85.590,-176.023,9.154,148.700
C08729=1178.824,412.301,-85.553,-176.022,9.153,148.700
C08730=1178.828,412.054,-85.518,-176.022,9.150,148.699
C08731=1178.833,411.806,-85.482,-176.022,9.149,148.699
C08732=1178.836,411.560,-85.445,-176.022,9.147,148.698
C08733=1178.840,411.312,-85.409,-176.022,9.145,148.697
C08734=1178.844,411.064,-85.374,-176.022,9.143,148.697
C08735=1178.848,410.817,-85.338,-176.022,9.140,148.696
C08736=1178.852,410.570,-85.301,-176.021,9.139,148.696
C08737=1178.855,410.322,-85.266,-176.022,9.136,148.695
C08738=1178.860,410.074,-85.229,-176.021,9.135,148.695
C08739=1178.863,409.827,-85.193,-176.021,9.132,148.694
C08740=1178.867,409.581,-85.158,-176.021,9.131,148.694
C08741=1178.872,409.333,-85.122,-176.021,9.128,148.693
C08742=1178.875,409.085,-85.086,-176.021,9.126,148.692
C08743=1178.879,408.838,-85.050,-176.021,9.125,148.692
C08744=1178.883,408.591,-85.014,-176.021,9.122,148.691
C08745=1178.887,408.343,-84.978,-176.020,9.121,148.691
C08746=1178.891,408.096,-84.942,-176.020,9.118,148.690
C08747=1178.895,407.848,-84.906,-176.020,9.116,148.689
C08748=1178.898,407.601,-84.870,-176.020,9.115,148.689
C08749=1178.903,407.353,-84.834,-176.020,9.112,148.688
C08750=1178.907,407.107,-84.798,-176.020,9.110,148.688
C08751=1178.910,406.859,-84.763,-176.019,9.108,148.687
C08752=1178.915,406.612,-84.727,-176.020,9.106,148.687
C08753=1178.918,406.364,-84.691,-176.020,9.103,148.686
C08754=1178.922,406.117,-84.654,-176.019,9.102,148.685
C08755=1178.926,405.869,-84.619,-176.019,9.099,148.685
C08756=1178.930,405.622,-84.583,-176.019,9.097,148.684
C08757=1178.934,405.374,-84.547,-176.019,9.095,148.683
C08758=1178.938,405.127,-84.512,-176.019,9.093,148.683
C08759=1178.942,404.880,-84.476,-176.019,9.090,148.682
C08760=1178.946,404.633,-84.439,-176.018,9.089,148.682
C08761=1178.950,404.385,-84.404,-176.018,9.086,148.681
C08762=1178.954,404.138,-84.368,-176.019,9.084,148.681
C08763=1178.958,403.890,-84.332,-176.018,9.081,148.680
C08764=1178.961,403.643,-84.296,-176.019,9.079,148.679
C08765=1178.966,403.396,-84.261,-176.018,9.077,148.679
C08766=1178.970,403.148,-84.225,-176.018,9.075,148.678
C08767=1178.974,402.901,-84.189,-176.018,9.073,148.677
C08768=1178.977,402.653,-84.154,-176.018,9.070,148.677
C08769=1178.981,402.406,-84.117,-176.018,9.068,148.676
C08770=1178.985,402.159,-84.081,-176.018,9.066,148.676
C08771=1178.989,401.911,-84.046,-176.018,9.064,148.675
C08772=1178.994,401.664,-84.010,-176.017,9.061,148.674
C08773=1178.997,401.416,-83.974,-176.018,9.059,148.674
C08774=1179.001,401.170,-83.938,-176.018,9.056,148.673
C08775=1179.005,400.922,-83.902,-176.018,9.054,148.673
C08776=1179.009,400.674,-83.866,-176.018,9.052,148.672
C08777=1179.012,400.427,-83.831,-176.018,9.049,148.671
C08778=1179.017,400.179,-83.795,-176.017,9.048,148.671
C08779=1179.021,399.932,-83.759,-176.017,9.045,148.670
C08780=1179.025,399.685,-83.724,-176.017,9.043,148.669
C08781=1179.028,399.438,-83.688,-176.017,9.040,148.669
C08782=1179.033,399.190,-83.651,-176.017,9.038,148.668
C08783=1179.036,398.942,-83.616,-176.017,9.035,148.667
C08784=1179.040,398.695,-83.580,-176.017,9.033,148.667
C08785=1179.045,398.448,-83.545,-176.017,9.030,148.666
C08786=1179.049,398.200,-83.509,-176.017,9.028,148.665
C08787=1179.052,397.953,-83.474,-176.017,9.025,148.665
C08788=1179.056,397.705,-83.438,-176.017,9.023,148.664
C08789=1179.060,397.458,-83.402,-176.018,9.020,148.663
C08790=1179.064,397.210,-83.366,-176.018,9.017,148.663
C08791=1179.068,396.964,-83.330,-176.018,9.015,148.662
C08792=1179.072,396.716,-83.294,-176.018,9.012,148.661
C08793=1179.076,396.469,-83.259,-176.018,9.010,148.661
C08794=1179.080,396.221,-83.223,-176.018,9.007,148.660
C08795=1179.083,395.974,-83.188,-176.018,9.005,148.660
C08796=1179.088,395.726,-83.152,-176.018,9.003,148.659
C08797=1179.092,395.479,-83.116,-176.018,8.999,148.658
C08798=1179.096,395.231,-83.081,-176.018,8.997,148.658
C08799=1179.099,394.984,-83.045,-176.018,8.994,148.657
C08800=1179.104,394.736,-83.009,-176.018,8.992,148.656
C08801=1179.108,394.489,-82.974,-176.018,8.990,148.656
C08802=1179.112,394.242,-82.938,-176.019,8.986,148.655
C08803=1179.115,393.994,-82.903,-176.019,8.984,148.654
C08804=1179.120,393.747,-82.867,-176.019,8.981,148.654
C08805=1179.123,393.499,-82.831,-176.019,8.979,148.653
C08806=1179.128,393.252,-82.796,-176.020,8.976,148.652
C08807=1179.131,393.005,-82.760,-176.019,8.973,148.652
C08808=1179.135,392.757,-82.725,-176.019,8.971,148.651
C08809=1179.139,392.509,-82.689,-176.020,8.967,148.650
C08810=1179.144,392.226,-82.648,-176.020,8.964,148.650
C08811=1179.148,391.941,-82.607,-176.020,8.961,148.649
C08812=1179.152,391.657,-82.566,-176.021,8.958,148.648
C08813=1179.157,391.373,-82.526,-176.021,8.955,148.647
C08814=1179.161,391.125,-82.490,-176.021,8.952,148.647
C08815=1179.164,390.878,-82.455,-176.022,8.949,148.646
C08816=1179.169,390.631,-82.419,-176.021,8.946,148.645
C08817=1179.173,390.383,-82.383,-176.022,8.943,148.645
C08818=1179.177,390.136,-82.348,-176.022,8.941,148.644
C08819=1179.180,389.888,-82.312,-176.023,8.937,148.643
C08820=1179.184,389.641,-82.277,-176.023,8.935,148.643
C08821=1179.188,389.394,-82.241,-176.023,8.932,148.642
C08822=1179.193,389.146,-82.205,-176.024,8.929,148.641
C08823=1179.197,388.898,-82.170,-176.024,8.926,148.641
C08824=1179.200,388.651,-82.135,-176.025,8.923,148.640
C08825=1179.205,388.404,-82.100,-176.025,8.920,148.639
C08826=1179.208,388.156,-82.064,-176.025,8.917,148.639
C08827=1179.212,387.909,-82.029,-176.026,8.914,148.638
C08828=1179.216,387.661,-81.993,-176.027,8.911,148.637
C08829=1179.221,387.414,-81.957,-176.027,8.909,148.637
C08830=1179.224,387.167,-81.922,-176.027,8.905,148.636
C08831=1179.228,386.919,-81.887,-176.028,8.902,148.636
C08832=1179.232,386.671,-81.851,-176.028,8.899,148.635
C08833=1179.236,386.424,-81.816,-176.029,8.896,148.634
C08834=1179.240,386.177,-81.781,-176.030,8.893,148.634
C08835=1179.244,385.929,-81.745,-176.030,8.890,148.633
C08836=1179.247,385.682,-81.710,-176.031,8.887,148.632
C08837=1179.252,385.434,-81.675,-176.031,8.883,148.632
C08838=1179.256,385.187,-81.639,-176.032,8.880,148.631
C08839=1179.260,384.939,-81.603,-176.033,8.877,148.630
C08840=1179.264,384.692,-81.568,-176.034,8.874,148.630
C08841=1179.268,384.444,-81.533,-176.034,8.871,148.629
C08842=1179.272,384.197,-81.498,-176.035,8.868,148.628
C08843=1179.276,383.950,-81.463,-176.036,8.865,148.628
C08844=1179.280,383.702,-81.427,-176.036,8.861,148.627
C08845=1179.284,383.454,-81.392,-176.037,8.858,148.626
C08846=1179.287,383.207,-81.357,-176.038,8.855,148.626
C08847=1179.292,382.960,-81.321,-176.038,8.852,148.625
C08848=1179.295,382.712,-81.286,-176.039,8.849,148.625
C08849=1179.299,382.464,-81.251,-176.040,8.846,148.624
C08850=1179.303,382.217,-81.216,-176.041,8.842,148.623
C08851=1179.307,381.970,-81.180,-176.041,8.839,148.623
C08852=1179.311,381.722,-81.146,-176.043,8.835,148.622
C08853=1179.315,381.475,-81.110,-176.044,8.832,148.622
C08854=1179.319,381.228,-81.075,-176.044,8.829,148.621
C08855=1179.323,380.979,-81.040,-176.045,8.826,148.620
C08856=1179.327,380.733,-81.005,-176.046,8.823,148.620
C08857=1179.331,380.485,-80.969,-176.047,8.819,148.619
C08858=1179.335,380.237,-80.934,-176.048,8.816,148.619
C08859=1179.339,379.990,-80.899,-176.049,8.813,148.618
C08860=1179.343,379.743,-80.864,-176.050,8.810,148.617
C08861=1179.347,379.495,-80.829,-176.051,8.806,148.617
C08862=1179.351,379.248,-80.794,-176.052,8.803,148.616
C08863=1179.355,379.000,-80.759,-176.053,8.800,148.616
C08864=1179.359,378.752,-80.723,-176.054,8.796,148.615
C08865=1179.363,378.505,-80.689,-176.055,8.793,148.614
C08866=1179.367,378.257,-80.653,-176.057,8.789,148.614
C08867=1179.371,378.010,-80.618,-176.057,8.786,148.613
C08868=1179.375,377.762,-80.583,-176.059,8.783,148.613
C08869=1179.379,377.515,-80.548,-176.060,8.779,148.612
C08870=1179.383,377.267,-80.513,-176.061,8.776,148.612
C08871=1179.387,377.020,-80.478,-176.062,8.772,148.611
C08872=1179.391,376.773,-80.444,-176.063,8.769,148.610
C08873=1179.394,376.525,-80.408,-176.065,8.765,148.610
C08874=1179.398,376.277,-80.373,-176.066,8.762,148.609
C08875=1179.403,376.030,-80.339,-176.067,8.758,148.609
C08876=1179.407,375.782,-80.303,-176.068,8.755,148.608
C08877=1179.411,375.535,-80.269,-176.070,8.751,148.608
C08878=1179.415,375.287,-80.233,-176.071,8.748,148.607
C08879=1179.419,375.039,-80.199,-176.072,8.744,148.607
C08880=1179.422,374.793,-80.164,-176.074,8.741,148.606
C08881=1179.426,374.545,-80.129,-176.075,8.738,148.606
C08882=1179.431,374.297,-80.095,-176.076,8.734,148.605
C08883=1179.435,374.050,-80.059,-176.077,8.731,148.605
C08884=1179.439,373.802,-80.025,-176.079,8.727,148.604
C08885=1179.443,373.555,-79.989,-176.080,8.724,148.603
C08886=1179.446,373.307,-79.955,-176.081,8.720,148.603
C08887=1179.451,373.060,-79.920,-176.083,8.717,148.602
C08888=1179.454,372.812,-79.885,-176.084,8.713,148.602
C08889=1179.459,372.565,-79.850,-176.086,8.710,148.601
C08890=1179.463,372.316,-79.816,-176.087,8.706,148.601
C08891=1179.467,372.069,-79.782,-176.089,8.703,148.600
C08892=1179.470,371.822,-79.746,-176.090,8.700,148.600
C08893=1179.475,371.574,-79.712,-176.092,8.696,148.599
C08894=1179.479,371.326,-79.677,-176.093,8.692,148.599
C08895=1179.482,371.080,-79.642,-176.095,8.688,148.598
C08896=1179.486,370.832,-79.607,-176.097,8.685,148.598
C08897=1179.491,370.584,-79.573,-176.098,8.682,148.597
C08898=1179.495,370.336,-79.538,-176.099,8.678,148.597
C08899=1179.499,370.089,-79.504,-176.101,8.674,148.596
C08900=1179.502,369.842,-79.469,-176.103,8.671,148.596
C08901=1179.507,369.594,-79.434,-176.104,8.668,148.596
C08902=1179.510,369.346,-79.400,-176.106,8.664,148.595
C08903=1179.515,369.099,-79.366,-176.107,8.660,148.595
C08904=1179.519,368.851,-79.331,-176.109,8.657,148.594
C08905=1179.523,368.603,-79.296,-176.111,8.653,148.594
C08906=1179.526,368.356,-79.261,-176.113,8.650,148.593
C08907=1179.531,368.109,-79.227,-176.115,8.646,148.593
C08908=1179.535,367.861,-79.192,-176.116,8.643,148.592
C08909=1179.539,367.614,-79.158,-176.117,8.639,148.592
C08910=1179.543,367.365,-79.123,-176.119,8.636,148.591
C08911=1179.546,367.118,-79.089,-176.121,8.632,148.591
C08912=1179.550,366.870,-79.055,-176.123,8.628,148.591
C08913=1179.555,366.623,-79.020,-176.125,8.625,148.590
C08914=1179.559,366.341,-78.981,-176.126,8.621,148.590
C08915=1179.564,366.060,-78.942,-176.129,8.617,148.589
C08916=1179.568,365.778,-78.903,-176.131,8.613,148.589
C08917=1179.573,365.496,-78.864,-176.133,8.609,148.588
C08918=1179.577,365.248,-78.829,-176.135,8.605,148.588
C08919=1179.581,365.001,-78.796,-176.137,8.601,148.587
C08920=1179.585,364.753,-78.761,-176.139,8.598,148.587
C08921=1179.589,364.506,-78.727,-176.140,8.594,148.587
C08922=1179.593,364.258,-78.692,-176.142,8.591,148.586
C08923=1179.597,364.011,-78.658,-176.144,8.587,148.586
C08924=1179.601,363.763,-78.624,-176.146,8.584,148.585
C08925=1179.605,363.515,-78.589,-176.148,8.580,148.585
C08926=1179.609,363.268,-78.555,-176.150,8.576,148.585
C08927=1179.612,363.020,-78.521,-176.152,8.573,148.584
C08928=1179.617,362.773,-78.486,-176.154,8.569,148.584
C08929=1179.621,362.525,-78.453,-176.156,8.566,148.583
C08930=1179.625,362.277,-78.418,-176.158,8.562,148.583
C08931=1179.629,362.030,-78.384,-176.160,8.559,148.583
C08932=1179.633,361.782,-78.350,-176.162,8.555,148.582
C08933=1179.637,361.534,-78.316,-176.164,8.552,148.582
C08934=1179.642,361.286,-78.282,-176.166,8.548,148.582
C08935=1179.645,361.039,-78.248,-176.168,8.545,148.581
C08936=1179.649,360.792,-78.214,-176.170,8.541,148.581
C08937=1179.653,360.544,-78.179,-176.172,8.538,148.581
C08938=1179.657,360.296,-78.146,-176.174,8.534,148.580
C08939=1179.661,360.048,-78.111,-176.176,8.531,148.580
C08940=1179.665,359.801,-78.078,-176.178,8.527,148.580
C08941=1179.670,359.553,-78.044,-176.180,8.524,148.579
C08942=1179.673,359.305,-78.010,-176.182,8.520,148.579
C08943=1179.677,359.058,-77.976,-176.185,8.516,148.579
C08944=1179.682,358.810,-77.942,-176.186,8.513,148.578
C08945=1179.685,358.562,-77.908,-176.189,8.509,148.578
C08946=1179.689,358.315,-77.874,-176.191,8.506,148.578
C08947=1179.694,358.067,-77.840,-176.193,8.502,148.577
C08948=1179.698,357.820,-77.806,-176.195,8.499,148.577
C08949=1179.701,357.572,-77.772,-176.197,8.495,148.577
C08950=1179.706,357.324,-77.738,-176.199,8.492,148.576
C08951=1179.710,357.077,-77.704,-176.201,8.488,148.576
C08952=1179.713,356.829,-77.671,-176.203,8.485,148.576
C08953=1179.718,356.581,-77.636,-176.206,8.481,148.576
C08954=1179.722,356.334,-77.603,-176.208,8.477,148.575
C08955=1179.726,356.086,-77.569,-176.210,8.474,148.575
C08956=1179.730,355.838,-77.535,-176.212,8.471,148.575
C08957=1179.734,355.591,-77.501,-176.214,8.467,148.574
C08958=1179.738,355.343,-77.468,-176.216,8.464,148.574
C08959=1179.742,355.096,-77.434,-176.219,8.461,148.574
C08960=1179.747,354.848,-77.401,-176.221,8.457,148.574
C08961=1179.750,354.599,-77.367,-176.223,8.454,148.573
C08962=1179.754,354.352,-77.333,-176.225,8.450,148.573
C08963=1179.758,354.104,-77.300,-176.228,8.446,148.573
C08964=1179.762,353.857,-77.266,-176.230,8.443,148.572
C08965=1179.767,353.609,-77.232,-176.232,8.439,148.572
C08966=1179.770,353.361,-77.199,-176.234,8.436,148.572
C08967=1179.774,353.114,-77.165,-176.237,8.433,148.572
C08968=1179.778,352.866,-77.132,-176.238,8.429,148.571
C08969=1179.782,352.618,-77.099,-176.241,8.426,148.571
C08970=1179.787,352.371,-77.064,-176.243,8.422,148.571
C08971=1179.791,352.123,-77.031,-176.245,8.419,148.570
C08972=1179.795,351.875,-76.998,-176.247,8.416,148.570
C08973=1179.799,351.628,-76.964,-176.249,8.412,148.570
C08974=1179.803,351.380,-76.930,-176.252,8.409,148.570
C08975=1179.807,351.132,-76.897,-176.254,8.405,148.569
C08976=1179.811,350.884,-76.864,-176.257,8.401,148.569
C08977=1179.816,350.637,-76.830,-176.259,8.398,148.569
C08978=1179.820,350.389,-76.797,-176.261,8.395,148.569
C08979=1179.823,350.141,-76.763,-176.263,8.391,148.568
C08980=1179.827,349.893,-76.730,-176.265,8.388,148.568
C08981=1179.831,349.645,-76.697,-176.267,8.385,148.568
C08982=1179.836,349.398,-76.664,-176.270,8.381,148.568
C08983=1179.839,349.151,-76.630,-176.272,8.378,148.567
C08984=1179.844,348.903,-76.597,-176.274,8.375,148.567
C08985=1179.848,348.655,-76.563,-176.277,8.371,148.567
C08986=1179.852,348.407,-76.530,-176.279,8.368,148.567
C08987=1179.856,348.160,-76.497,-176.281,8.365,148.567
C08988=1179.860,347.912,-76.464,-176.283,8.361,148.566
C08989=1179.864,347.663,-76.430,-176.286,8.357,148.566
C08990=1179.868,347.416,-76.397,-176.288,8.354,148.566
C08991=1179.872,347.168,-76.364,-176.291,8.351,148.566
C08992=1179.876,346.920,-76.331,-176.293,8.347,148.565
C08993=1179.880,346.673,-76.298,-176.295,8.344,148.565
C08994=1179.884,346.425,-76.265,-176.297,8.340,148.565
C08995=1179.889,346.177,-76.231,-176.299,8.337,148.565
C08996=1179.893,345.929,-76.198,-176.302,8.334,148.564
C08997=1179.897,345.682,-76.165,-176.304,8.330,148.564
C08998=1179.901,345.434,-76.132,-176.306,8.327,148.564
C08999=1179.905,345.186,-76.099,-176.308,8.324,148.564
C09000=1179.909,344.938,-76.066,-176.311,8.320,148.563
C09001=1179.913,344.691,-76.033,-176.313,8.317,148.563
C09002=1179.917,344.443,-75.999,-176.316,8.314,148.563
C09003=1179.922,344.195,-75.967,-176.318,8.311,148.563
C09004=1179.926,343.947,-75.934,-176.320,8.308,148.563
C09005=1179.930,343.699,-75.901,-176.322,8.304,148.563
C09006=1179.934,343.452,-75.868,-176.325,8.301,148.562
C09007=1179.938,343.204,-75.835,-176.327,8.298,148.562
C09008=1179.942,342.956,-75.802,-176.330,8.293,148.562
C09009=1179.946,342.708,-75.769,-176.332,8.290,148.562
C09010=1179.950,342.460,-75.736,-176.334,8.287,148.561
C09011=1179.955,342.212,-75.703,-176.337,8.284,148.561
C09012=1179.959,341.965,-75.670,-176.339,8.280,148.561
C09013=1179.962,341.717,-75.638,-176.341,8.277,148.561
C09014=1179.967,341.469,-75.605,-176.344,8.274,148.561
C09015=1179.971,341.221,-75.572,-176.346,8.271,148.561
C09016=1179.975,340.974,-75.539,-176.348,8.267,148.560
C09017=1179.980,340.726,-75.506,-176.351,8.264,148.560
C09018=1179.984,340.447,-75.470,-176.353,8.261,148.560
C09019=1179.989,340.168,-75.432,-176.356,8.257,148.560
C09020=1179.993,339.889,-75.396,-176.358,8.253,148.559
C09021=1179.997,339.610,-75.359,-176.361,8.249,148.559
C09022=1180.002,339.362,-75.326,-176.364,8.246,148.559
C09023=1180.006,339.114,-75.293,-176.366,8.243,148.559
C09024=1180.010,338.865,-75.261,-176.368,8.239,148.559
C09025=1180.014,338.619,-75.229,-176.370,8.236,148.559
C09026=1180.018,338.371,-75.195,-176.373,8.233,148.559
C09027=1180.023,338.123,-75.163,-176.375,8.230,148.558
C09028=1180.026,337.875,-75.130,-176.378,8.226,148.558
C09029=1180.031,337.627,-75.098,-176.380,8.223,148.558
C09030=1180.035,337.379,-75.065,-176.382,8.220,148.558
C09031=1180.039,337.131,-75.033,-176.385,8.217,148.558
C09032=1180.043,336.883,-75.000,-176.387,8.214,148.557
C09033=1180.048,336.636,-74.968,-176.389,8.210,148.557
C09034=1180.051,336.388,-74.935,-176.392,8.207,148.557
C09035=1180.056,336.140,-74.903,-176.394,8.204,148.557
C09036=1180.060,335.892,-74.870,-176.397,8.201,148.557
C09037=1180.063,335.644,-74.838,-176.399,8.197,148.557
C09038=1180.068,335.396,-74.805,-176.401,8.194,148.556
C09039=1180.072,335.149,-74.773,-176.404,8.191,148.556
C09040=1180.076,334.901,-74.741,-176.406,8.188,148.556
C09041=1180.081,334.652,-74.708,-176.408,8.184,148.556
C09042=1180.084,334.405,-74.676,-176.411,8.181,148.556
C09043=1180.089,334.157,-74.643,-176.413,8.178,148.556
C09044=1180.092,333.909,-74.611,-176.416,8.175,148.556
C09045=1180.097,333.662,-74.579,-176.418,8.171,148.555
C09046=1180.101,333.414,-74.547,-176.421,8.168,148.555
C09047=1180.105,333.165,-74.514,-176.423,8.165,148.555
C09048=1180.109,332.918,-74.482,-176.425,8.162,148.555
C09049=1180.114,332.670,-74.450,-176.428,8.159,148.555
C09050=1180.117,332.422,-74.418,-176.430,8.156,148.555
C09051=1180.122,332.174,-74.385,-176.432,8.152,148.555
C09052=1180.125,331.926,-74.353,-176.435,8.149,148.555
C09053=1180.130,331.679,-74.321,-176.437,8.146,148.554
C09054=1180.134,331.431,-74.289,-176.440,8.143,148.554
C09055=1180.138,331.182,-74.256,-176.442,8.140,148.554
C09056=1180.142,330.934,-74.225,-176.445,8.136,148.554
C09057=1180.147,330.687,-74.192,-176.447,8.133,148.554
C09058=1180.151,330.439,-74.160,-176.450,8.130,148.554
C09059=1180.155,330.191,-74.128,-176.452,8.127,148.554
C09060=1180.159,329.943,-74.096,-176.454,8.123,148.553
C09061=1180.163,329.696,-74.064,-176.457,8.120,148.553
C09062=1180.167,329.447,-74.032,-176.459,8.117,148.553
C09063=1180.171,329.199,-74.000,-176.462,8.114,148.553
C09064=1180.176,328.951,-73.968,-176.464,8.111,148.553
C09065=1180.180,328.703,-73.936,-176.466,8.107,148.553
C09066=1180.184,328.455,-73.904,-176.469,8.104,148.553
C09067=1180.189,328.208,-73.872,-176.471,8.101,148.552
C09068=1180.192,327.960,-73.840,-176.474,8.098,148.552
C09069=1180.196,327.712,-73.808,-176.476,8.095,148.552
C09070=1180.201,327.463,-73.776,-176.479,8.091,148.552
C09071=1180.205,327.216,-73.745,-176.481,8.088,148.552
C09072=1180.209,326.968,-73.713,-176.484,8.085,148.552
C09073=1180.214,326.720,-73.681,-176.486,8.082,148.552
C09074=1180.217,326.472,-73.649,-176.488,8.079,148.552
C09075=1180.221,326.224,-73.617,-176.491,8.076,148.552
C09076=1180.226,325.977,-73.585,-176.493,8.073,148.551
C09077=1180.230,325.729,-73.553,-176.496,8.070,148.551
C09078=1180.233,325.480,-73.521,-176.498,8.066,148.551
C09079=1180.238,325.233,-73.490,-176.501,8.063,148.551
C09080=1180.243,324.984,-73.458,-176.503,8.060,148.551
C09081=1180.246,324.736,-73.426,-176.506,8.057,148.551
C09082=1180.251,324.489,-73.395,-176.508,8.054,148.551
C09083=1180.254,324.241,-73.363,-176.511,8.050,148.551
C09084=1180.259,323.993,-73.331,-176.513,8.047,148.551
C09085=1180.263,323.745,-73.299,-176.516,8.044,148.550
C09086=1180.267,323.496,-73.268,-176.518,8.041,148.550
C09087=1180.271,323.249,-73.236,-176.521,8.038,148.550
C09088=1180.275,323.001,-73.204,-176.523,8.035,148.550
C09089=1180.279,322.754,-73.173,-176.526,8.031,148.550
C09090=1180.284,322.505,-73.141,-176.528,8.028,148.550
C09091=1180.288,322.257,-73.109,-176.531,8.025,148.550
C09092=1180.292,322.009,-73.078,-176.533,8.022,148.550
C09093=1180.296,321.761,-73.047,-176.535,8.020,148.550
C09094=1180.300,321.513,-73.015,-176.538,8.017,148.550
C09095=1180.304,321.265,-72.983,-176.540,8.013,148.550
C09096=1180.309,321.017,-72.953,-176.543,8.010,148.550
C09097=1180.312,320.769,-72.921,-176.545,8.007,148.550
C09098=1180.317,320.522,-72.889,-176.548,8.004,148.549
C09099=1180.321,320.273,-72.858,-176.550,8.001,148.549
C09100=1180.326,320.026,-72.826,-176.553,7.998,148.549
C09101=1180.330,319.777,-72.795,-176.555,7.995,148.549
C09102=1180.334,319.530,-72.764,-176.558,7.991,148.549
C09103=1180.338,319.281,-72.732,-176.560,7.988,148.549
C09104=1180.342,319.034,-72.701,-176.563,7.985,148.549
C09105=1180.346,318.786,-72.669,-176.565,7.982,148.549
C09106=1180.351,318.538,-72.638,-176.568,7.979,148.549
C09107=1180.354,318.290,-72.606,-176.570,7.976,148.549
C09108=1180.359,318.042,-72.576,-176.573,7.973,148.549
C09109=1180.363,317.793,-72.545,-176.575,7.969,148.548
C09110=1180.367,317.546,-72.513,-176.578,7.966,148.548
C09111=1180.371,317.297,-72.482,-176.580,7.963,148.548
C09112=1180.376,317.050,-72.450,-176.582,7.961,148.548
C09113=1180.380,316.801,-72.419,-176.585,7.958,148.548
C09114=1180.384,316.554,-72.388,-176.587,7.955,148.548
C09115=1180.388,316.305,-72.357,-176.590,7.952,148.548
C09116=1180.393,316.057,-72.326,-176.592,7.948,148.548
C09117=1180.396,315.809,-72.294,-176.595,7.945,148.548
C09118=1180.401,315.561,-72.263,-176.598,7.942,148.548
C09119=1180.406,315.313,-72.233,-176.600,7.939,148.548
C09120=1180.409,315.065,-72.201,-176.603,7.936,148.548
C09121=1180.413,314.817,-72.171,-176.605,7.933,148.548
C09122=1180.418,314.541,-72.135,-176.608,7.930,148.548
C09123=1180.422,314.264,-72.101,-176.611,7.926,148.548
C09124=1180.428,313.987,-72.066,-176.614,7.923,148.548
C09125=1180.432,313.710,-72.032,-176.616,7.920,148.547
C09126=1180.436,313.462,-72.001,-176.619,7.917,148.547
C09127=1180.441,313.214,-71.970,-176.622,7.914,148.547
C09128=1180.445,312.966,-71.938,-176.624,7.910,148.547
C09129=1180.449,312.718,-71.907,-176.627,7.907,148.547
C09130=1180.453,312.471,-71.877,-176.629,7.904,148.547
C09131=1180.457,312.222,-71.846,-176.632,7.901,148.547
C09132=1180.462,311.974,-71.815,-176.634,7.898,148.547
C09133=1180.466,311.726,-71.785,-176.637,7.895,148.547
C09134=1180.470,311.478,-71.753,-176.639,7.892,148.547
C09135=1180.474,311.230,-71.723,-176.642,7.889,148.547
C09136=1180.479,310.982,-71.692,-176.644,7.886,148.547
C09137=1180.483,310.734,-71.661,-176.646,7.883,148.547
C09138=1180.487,310.486,-71.630,-176.649,7.880,148.547
C09139=1180.491,310.238,-71.600,-176.652,7.877,148.547
C09140=1180.495,309.989,-71.569,-176.654,7.874,148.547
C09141=1180.500,309.742,-71.538,-176.657,7.871,148.547
